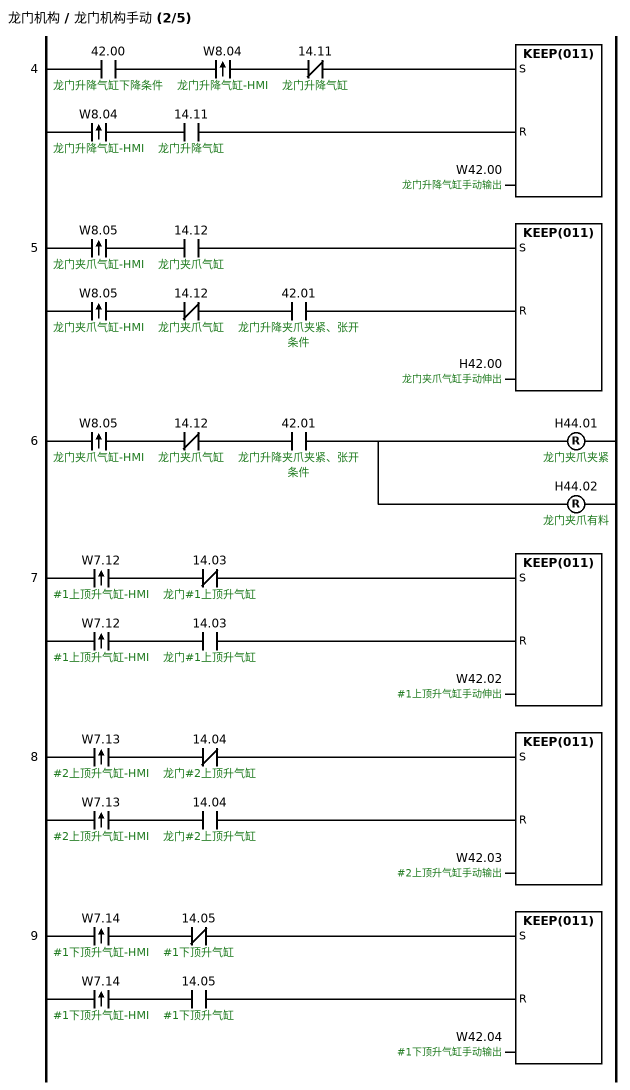
; [picture p377: 龙门机构 / 龙门机构手动, rungs 4-9]
; rung 4
LD 42.00  ; 龙门升降气缸下降条件
@AND W8.04  ; 龙门升降气缸-HMI
ANDNOT 14.11  ; 龙门升降气缸
@LD W8.04  ; 龙门升降气缸-HMI
AND 14.11  ; 龙门升降气缸
KEEP(011) W42.00  ; 龙门升降气缸手动输出
; rung 5
@LD W8.05  ; 龙门夹爪气缸-HMI
AND 14.12  ; 龙门夹爪气缸
@LD W8.05  ; 龙门夹爪气缸-HMI
ANDNOT 14.12  ; 龙门夹爪气缸
AND 42.01  ; 龙门升降夹爪夹紧、张开条件
KEEP(011) H42.00  ; 龙门夹爪气缸手动伸出
; rung 6
@LD W8.05  ; 龙门夹爪气缸-HMI
ANDNOT 14.12  ; 龙门夹爪气缸
AND 42.01  ; 龙门升降夹爪夹紧、张开条件
RSET H44.01  ; 龙门夹爪夹紧
RSET H44.02  ; 龙门夹爪有料
; rung 7
@LD W7.12  ; #1上顶升气缸-HMI
ANDNOT 14.03  ; 龙门#1上顶升气缸
@LD W7.12  ; #1上顶升气缸-HMI
AND 14.03  ; 龙门#1上顶升气缸
KEEP(011) W42.02  ; #1上顶升气缸手动伸出
; rung 8
@LD W7.13  ; #2上顶升气缸-HMI
ANDNOT 14.04  ; 龙门#2上顶升气缸
@LD W7.13  ; #2上顶升气缸-HMI
AND 14.04  ; 龙门#2上顶升气缸
KEEP(011) W42.03  ; #2上顶升气缸手动输出
; rung 9
@LD W7.14  ; #1下顶升气缸-HMI
ANDNOT 14.05  ; #1下顶升气缸
@LD W7.14  ; #1下顶升气缸-HMI
AND 14.05  ; #1下顶升气缸
KEEP(011) W42.04  ; #1下顶升气缸手动输出

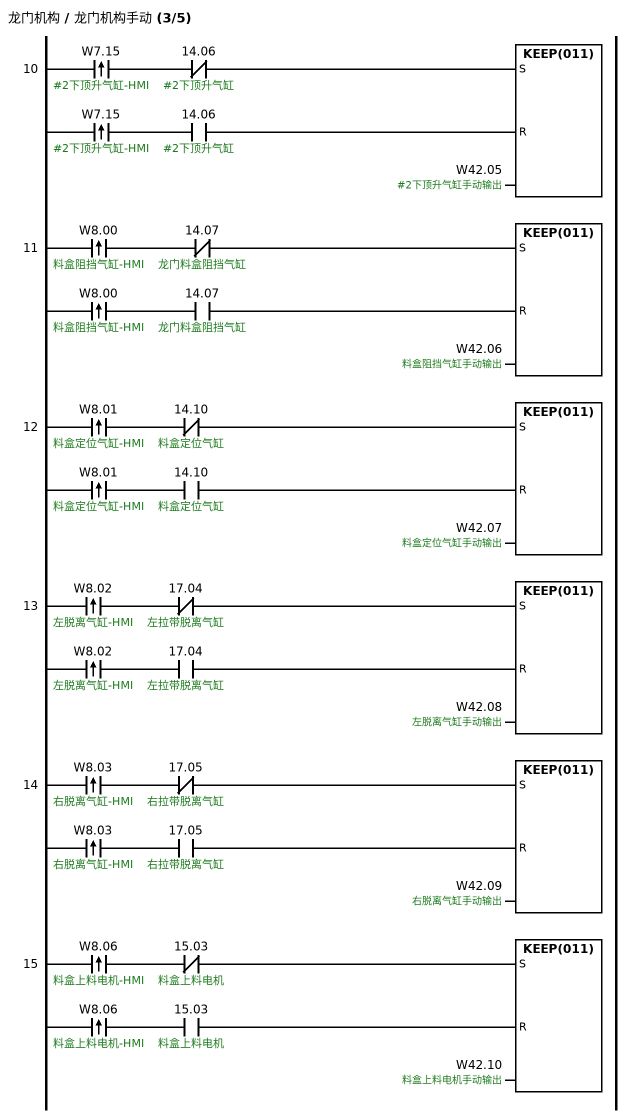
; rung 10
@LD W7.15  ; #2下顶升气缸-HMI
ANDNOT 14.06  ; #2下顶升气缸
@LD W7.15  ; #2下顶升气缸-HMI
AND 14.06  ; #2下顶升气缸
KEEP(011) W42.05  ; #2下顶升气缸手动输出
; rung 11
@LD W8.00  ; 料盒阻挡气缸-HMI
ANDNOT 14.07  ; 龙门料盒阻挡气缸
@LD W8.00  ; 料盒阻挡气缸-HMI
AND 14.07  ; 龙门料盒阻挡气缸
KEEP(011) W42.06  ; 料盒阻挡气缸手动输出
; rung 12
@LD W8.01  ; 料盒定位气缸-HMI
ANDNOT 14.10  ; 料盒定位气缸
@LD W8.01  ; 料盒定位气缸-HMI
AND 14.10  ; 料盒定位气缸
KEEP(011) W42.07  ; 料盒定位气缸手动输出
; rung 13
@LD W8.02  ; 左脱离气缸-HMI
ANDNOT 17.04  ; 左拉带脱离气缸
@LD W8.02  ; 左脱离气缸-HMI
AND 17.04  ; 左拉带脱离气缸
KEEP(011) W42.08  ; 左脱离气缸手动输出
; rung 14
@LD W8.03  ; 右脱离气缸-HMI
ANDNOT 17.05  ; 右拉带脱离气缸
@LD W8.03  ; 右脱离气缸-HMI
AND 17.05  ; 右拉带脱离气缸
KEEP(011) W42.09  ; 右脱离气缸手动输出
; rung 15
@LD W8.06  ; 料盒上料电机-HMI
ANDNOT 15.03  ; 料盒上料电机
@LD W8.06  ; 料盒上料电机-HMI
AND 15.03  ; 料盒上料电机
KEEP(011) W42.10  ; 料盒上料电机手动输出

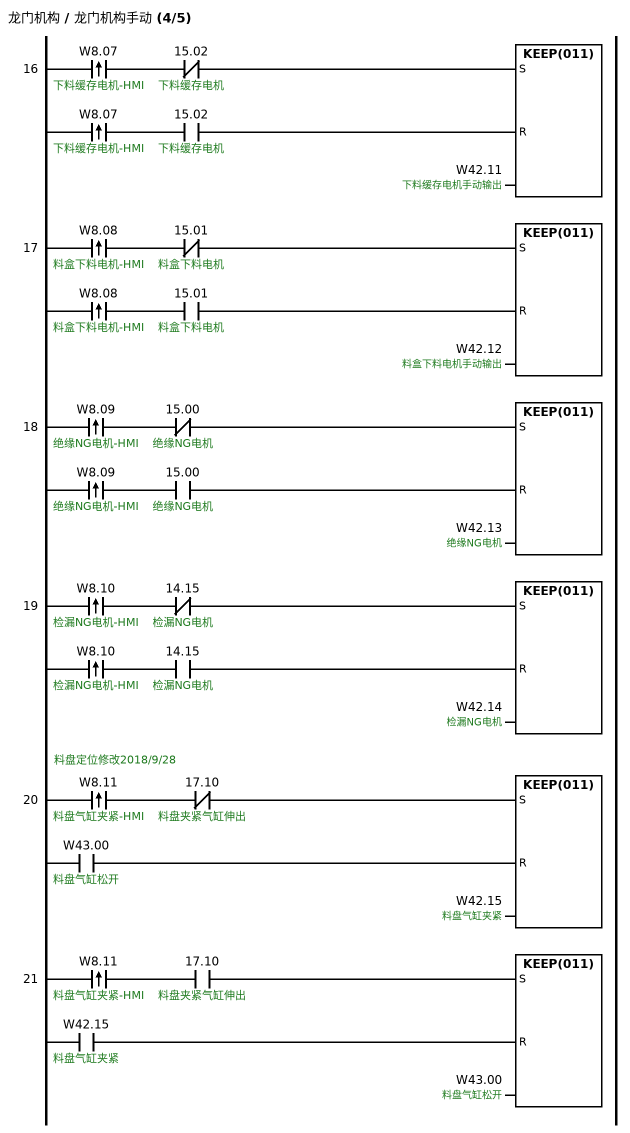
; rung 16
@LD W8.07  ; 下料缓存电机-HMI
ANDNOT 15.02  ; 下料缓存电机
@LD W8.07  ; 下料缓存电机-HMI
AND 15.02  ; 下料缓存电机
KEEP(011) W42.11  ; 下料缓存电机手动输出
; rung 17
@LD W8.08  ; 料盒下料电机-HMI
ANDNOT 15.01  ; 料盒下料电机
@LD W8.08  ; 料盒下料电机-HMI
AND 15.01  ; 料盒下料电机
KEEP(011) W42.12  ; 料盒下料电机手动输出
; rung 18
@LD W8.09  ; 绝缘NG电机-HMI
ANDNOT 15.00  ; 绝缘NG电机
@LD W8.09  ; 绝缘NG电机-HMI
AND 15.00  ; 绝缘NG电机
KEEP(011) W42.13  ; 绝缘NG电机
; rung 19
@LD W8.10  ; 检漏NG电机-HMI
ANDNOT 14.15  ; 检漏NG电机
@LD W8.10  ; 检漏NG电机-HMI
AND 14.15  ; 检漏NG电机
KEEP(011) W42.14  ; 检漏NG电机
; rung 20: 料盘定位修改2018/9/28
@LD W8.11  ; 料盘气缸夹紧-HMI
ANDNOT 17.10  ; 料盘夹紧气缸伸出
LD W43.00  ; 料盘气缸松开
KEEP(011) W42.15  ; 料盘气缸夹紧
; rung 21
@LD W8.11  ; 料盘气缸夹紧-HMI
AND 17.10  ; 料盘夹紧气缸伸出
LD W42.15  ; 料盘气缸夹紧
KEEP(011) W43.00  ; 料盘气缸松开

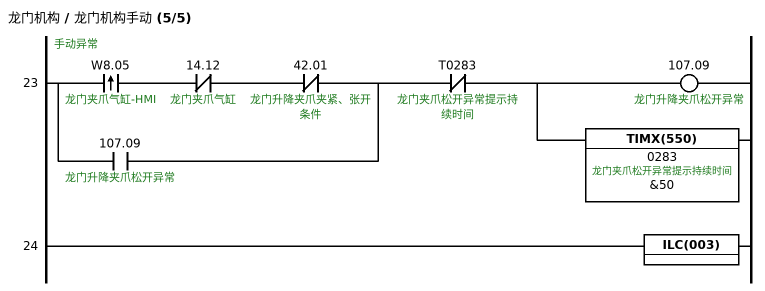
; rung 23: 手动异常
@LD W8.05  ; 龙门夹爪气缸-HMI
ANDNOT 14.12  ; 龙门夹爪气缸
ANDNOT 42.01  ; 龙门升降夹爪夹紧、张开条件
OR 107.09  ; 龙门升降夹爪松开异常
ANDNOT T0283  ; 龙门夹爪松开异常提示持续时间
OUT 107.09  ; 龙门升降夹爪松开异常
TIMX(550) 0283 &50  ; 龙门夹爪松开异常提示持续时间
; rung 24
ILC(003)

### Section 上料盒自动

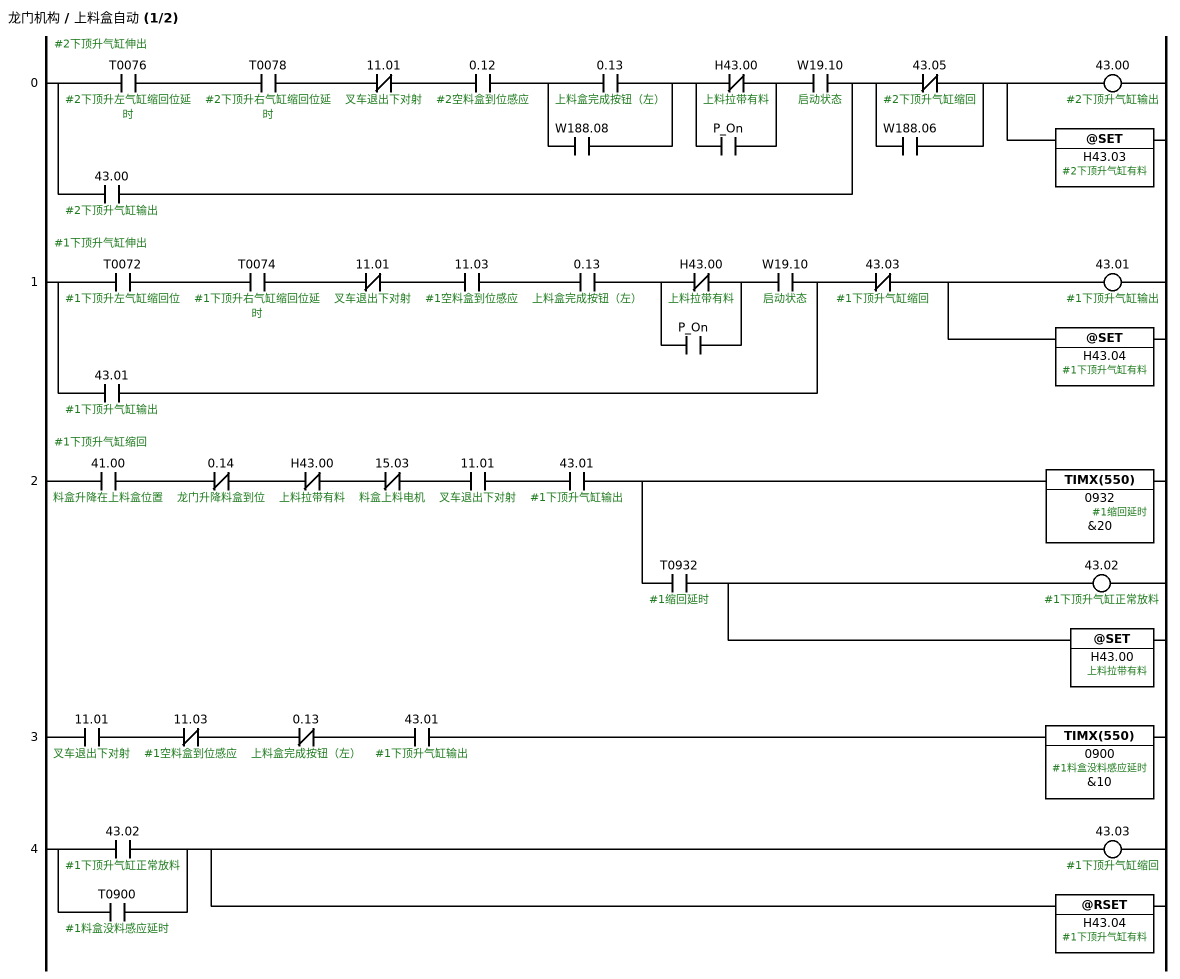
; rung 0: #2下顶升气缸伸出
LD T0076  ; #2下顶升左气缸缩回位延时
AND T0078  ; #2下顶升右气缸缩回位延时
ANDNOT 11.01  ; 叉车退出下对射
AND 0.12  ; #2空料盒到位感应
LD 0.13  ; 上料盒完成按钮（左）
OR W188.08
ANDLD
LDNOT H43.00  ; 上料拉带有料
OR P_On
ANDLD
AND W19.10  ; 启动状态
OR 43.00  ; #2下顶升气缸输出
LDNOT 43.05  ; #2下顶升气缸缩回
OR W188.06
ANDLD
OUT 43.00  ; #2下顶升气缸输出
@SET H43.03  ; #2下顶升气缸有料
; rung 1: #1下顶升气缸伸出
LD T0072  ; #1下顶升左气缸缩回位
AND T0074  ; #1下顶升右气缸缩回位延时
ANDNOT 11.01  ; 叉车退出下对射
AND 11.03  ; #1空料盒到位感应
AND 0.13  ; 上料盒完成按钮（左）
LDNOT H43.00  ; 上料拉带有料
OR P_On
ANDLD
AND W19.10  ; 启动状态
OR 43.01  ; #1下顶升气缸输出
ANDNOT 43.03  ; #1下顶升气缸缩回
OUT 43.01  ; #1下顶升气缸输出
@SET H43.04  ; #1下顶升气缸有料
; rung 2: #1下顶升气缸缩回
LD 41.00  ; 料盒升降在上料盒位置
ANDNOT 0.14  ; 龙门升降料盒到位
ANDNOT H43.00  ; 上料拉带有料
ANDNOT 15.03  ; 料盒上料电机
AND 11.01  ; 叉车退出下对射
AND 43.01  ; #1下顶升气缸输出
TIMX(550) 0932 &20  ; #1缩回延时
AND T0932  ; #1缩回延时
OUT 43.02  ; #1下顶升气缸正常放料
@SET H43.00  ; 上料拉带有料
; rung 3
LD 11.01  ; 叉车退出下对射
ANDNOT 11.03  ; #1空料盒到位感应
ANDNOT 0.13  ; 上料盒完成按钮（左）
AND 43.01  ; #1下顶升气缸输出
TIMX(550) 0900 &10  ; #1料盒没料感应延时
; rung 4
LD 43.02  ; #1下顶升气缸正常放料
OR T0900  ; #1料盒没料感应延时
OUT 43.03  ; #1下顶升气缸缩回
@RSET H43.04  ; #1下顶升气缸有料

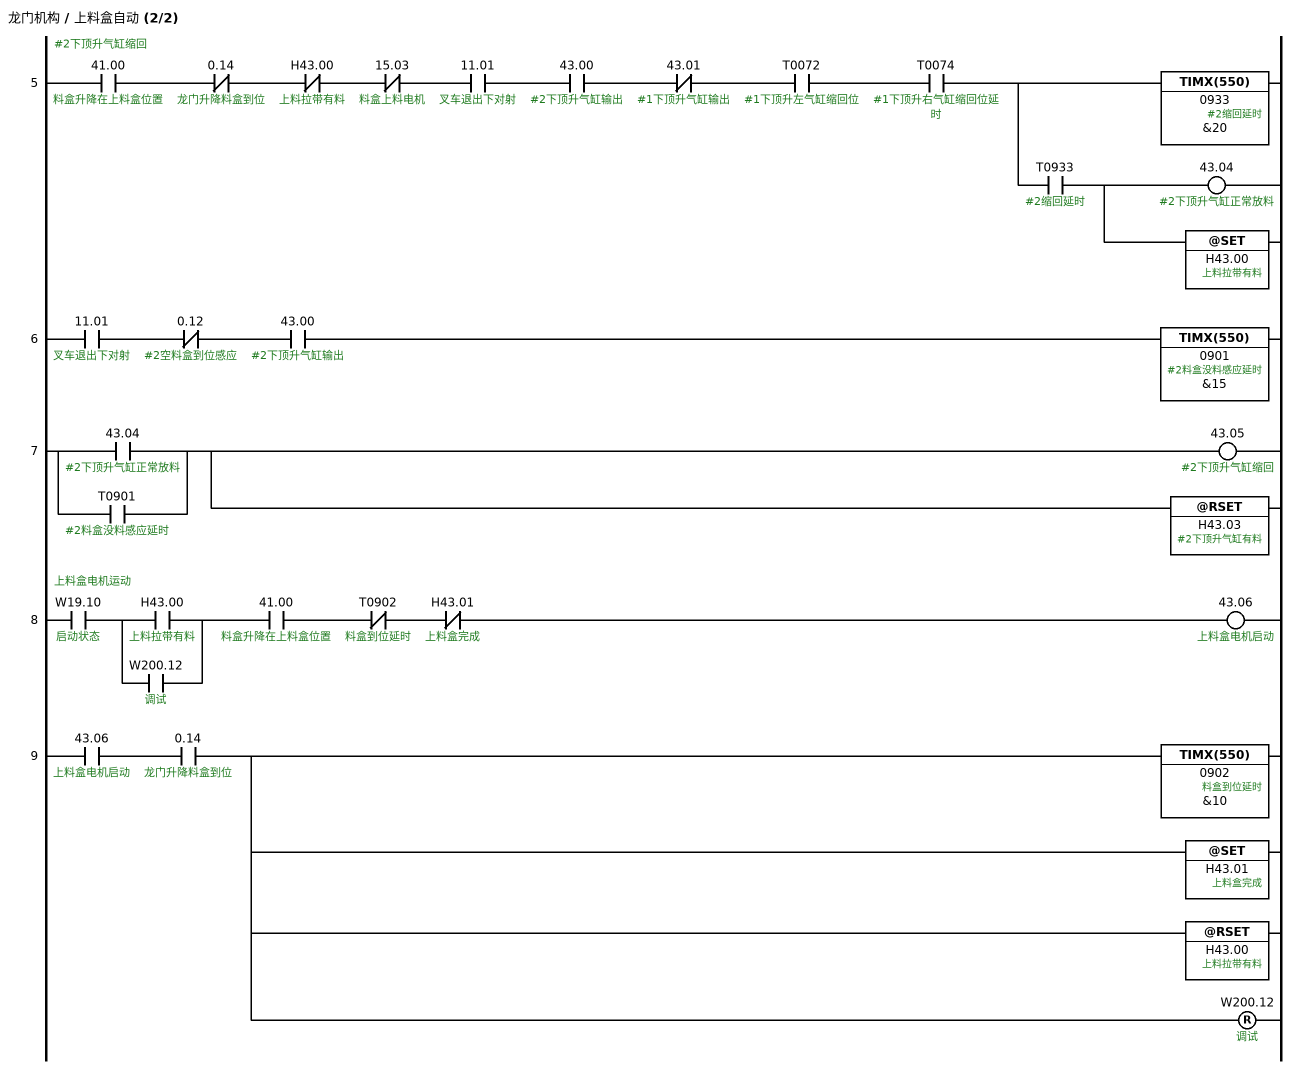
; rung 5: #2下顶升气缸缩回
LD 41.00  ; 料盒升降在上料盒位置
ANDNOT 0.14  ; 龙门升降料盒到位
ANDNOT H43.00  ; 上料拉带有料
ANDNOT 15.03  ; 料盒上料电机
AND 11.01  ; 叉车退出下对射
AND 43.00  ; #2下顶升气缸输出
ANDNOT 43.01  ; #1下顶升气缸输出
AND T0072  ; #1下顶升左气缸缩回位
AND T0074  ; #1下顶升右气缸缩回位延时
TIMX(550) 0933 &20  ; #2缩回延时
AND T0933  ; #2缩回延时
OUT 43.04  ; #2下顶升气缸正常放料
@SET H43.00  ; 上料拉带有料
; rung 6
LD 11.01  ; 叉车退出下对射
ANDNOT 0.12  ; #2空料盒到位感应
AND 43.00  ; #2下顶升气缸输出
TIMX(550) 0901 &15  ; #2料盒没料感应延时
; rung 7
LD 43.04  ; #2下顶升气缸正常放料
OR T0901  ; #2料盒没料感应延时
OUT 43.05  ; #2下顶升气缸缩回
@RSET H43.03  ; #2下顶升气缸有料
; rung 8: 上料盒电机运动
LD W19.10  ; 启动状态
LD H43.00  ; 上料拉带有料
OR W200.12  ; 调试
ANDLD
AND 41.00  ; 料盒升降在上料盒位置
ANDNOT T0902  ; 料盒到位延时
ANDNOT H43.01  ; 上料盒完成
OUT 43.06  ; 上料盒电机启动
; rung 9
LD 43.06  ; 上料盒电机启动
AND 0.14  ; 龙门升降料盒到位
TIMX(550) 0902 &10  ; 料盒到位延时
@SET H43.01  ; 上料盒完成
@RSET H43.00  ; 上料拉带有料
RSET W200.12  ; 调试

### Section 龙门机械手自动取放料

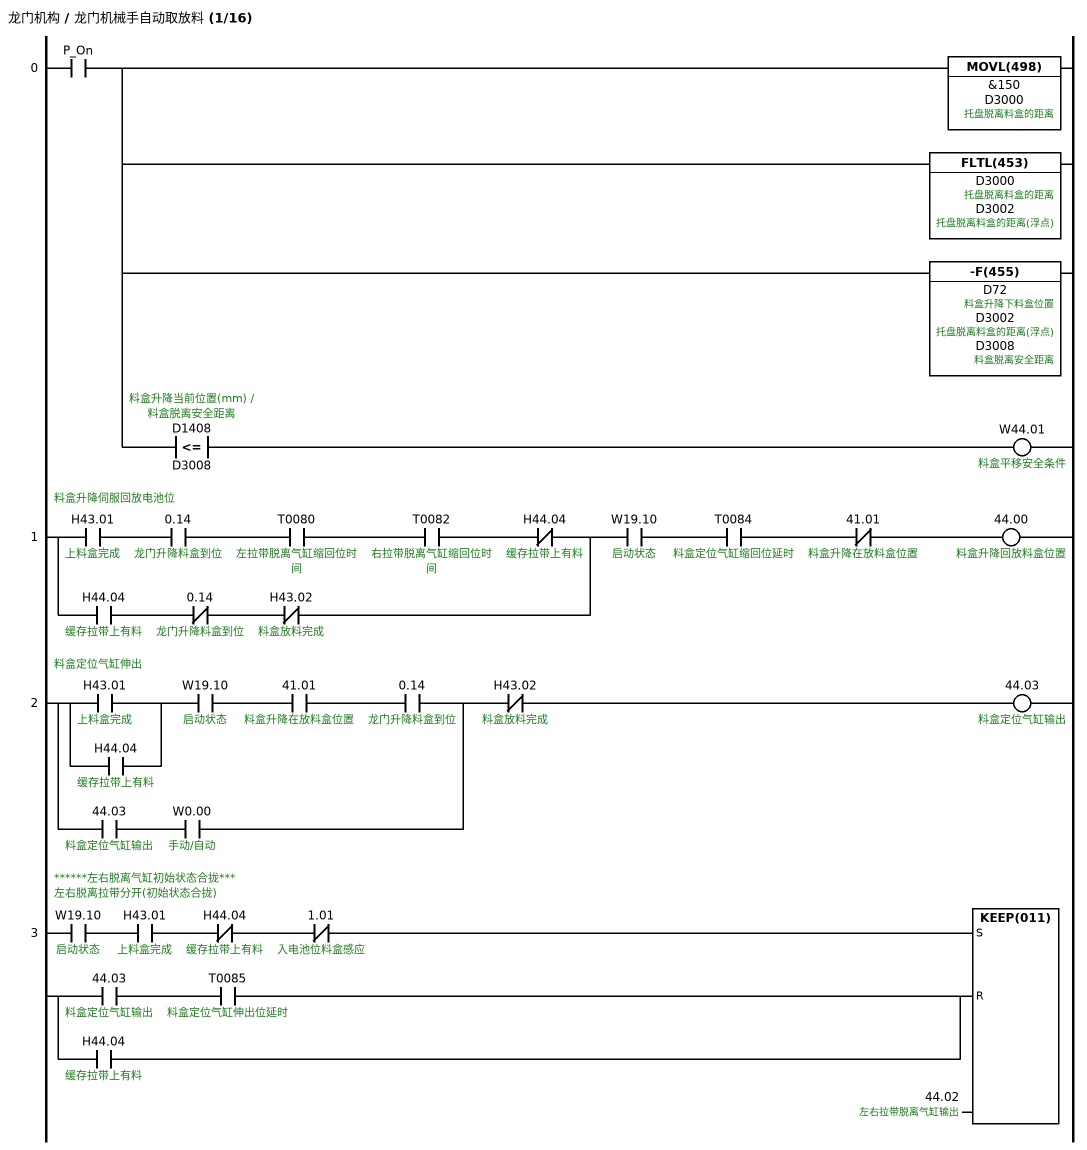
; rung 0
LD P_On
MOVL(498) &150 D3000  ; 托盘脱离料盒的距离
FLTL(453) D3000 D3002  ; 托盘脱离料盒的距离, 托盘脱离料盒的距离(浮点)
-F(455) D72 D3002 D3008  ; 料盒升降下料盒位置, 托盘脱离料盒的距离(浮点), 料盒脱离安全距离
AND<=F(332) D1408 D3008  ; 料盒升降当前位置(mm), 料盒脱离安全距离
OUT W44.01  ; 料盒平移安全条件
; rung 1: 料盒升降伺服回放电池位
LD H43.01  ; 上料盒完成
AND 0.14  ; 龙门升降料盒到位
AND T0080  ; 左拉带脱离气缸缩回位时间
AND T0082  ; 右拉带脱离气缸缩回位时间
ANDNOT H44.04  ; 缓存拉带上有料
LD H44.04  ; 缓存拉带上有料
ANDNOT 0.14  ; 龙门升降料盒到位
ANDNOT H43.02  ; 料盒放料完成
ORLD
AND W19.10  ; 启动状态
AND T0084  ; 料盒定位气缸缩回位延时
ANDNOT 41.01  ; 料盒升降在放料盒位置
OUT 44.00  ; 料盒升降回放料盒位置
; rung 2: 料盒定位气缸伸出
LD H43.01  ; 上料盒完成
OR H44.04  ; 缓存拉带上有料
AND W19.10  ; 启动状态
AND 41.01  ; 料盒升降在放料盒位置
AND 0.14  ; 龙门升降料盒到位
LD 44.03  ; 料盒定位气缸输出
AND W0.00  ; 手动/自动
ORLD
ANDNOT H43.02  ; 料盒放料完成
OUT 44.03  ; 料盒定位气缸输出
; rung 3: ******左右脱离气缸初始状态合拢*** / 左右脱离拉带分开(初始状态合拢)
LD W19.10  ; 启动状态
AND H43.01  ; 上料盒完成
ANDNOT H44.04  ; 缓存拉带上有料
ANDNOT 1.01  ; 入电池位料盒感应
LD 44.03  ; 料盒定位气缸输出
AND T0085  ; 料盒定位气缸伸出位延时
OR H44.04  ; 缓存拉带上有料
KEEP(011) 44.02  ; 左右拉带脱离气缸输出

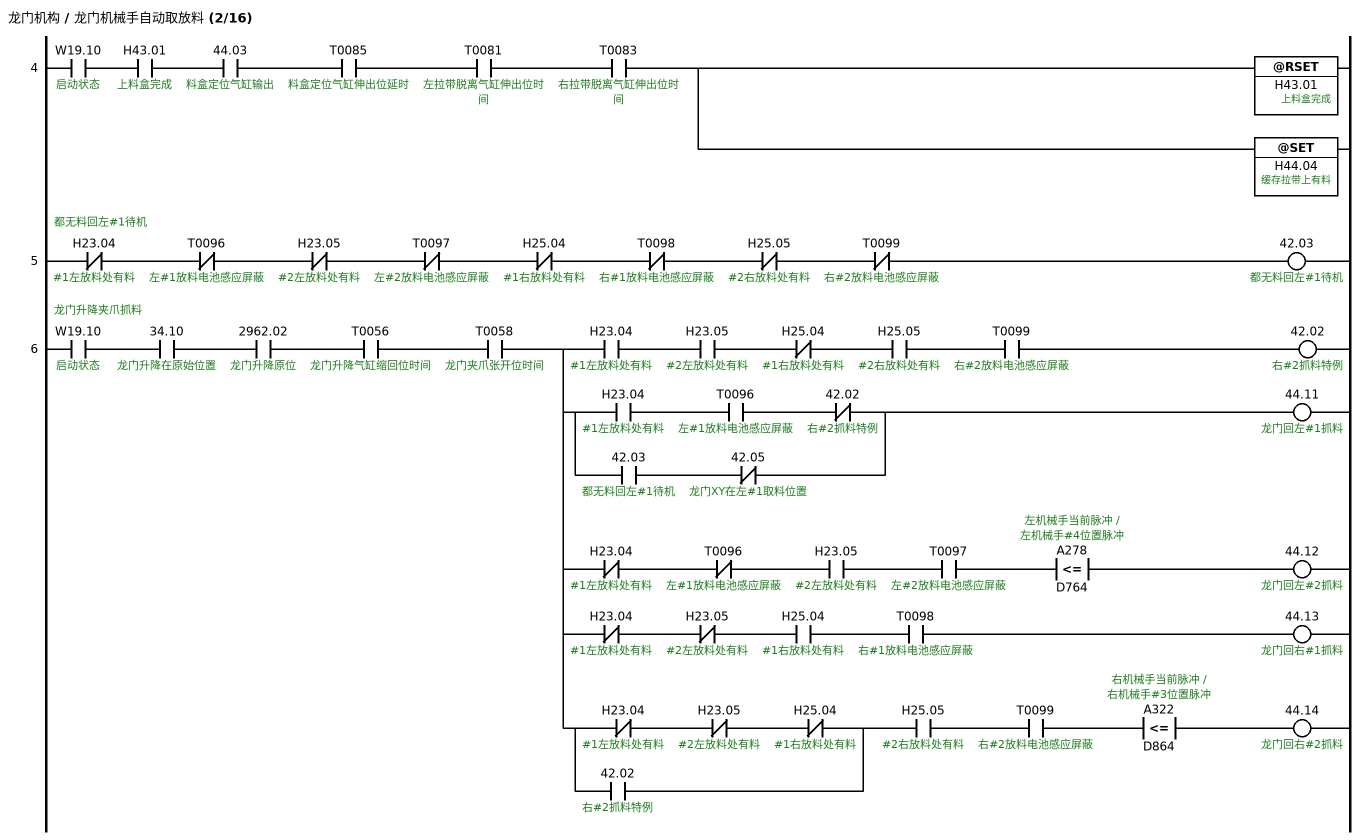
; rung 4
LD W19.10  ; 启动状态
AND H43.01  ; 上料盒完成
AND 44.03  ; 料盒定位气缸输出
AND T0085  ; 料盒定位气缸伸出位延时
AND T0081  ; 左拉带脱离气缸伸出位时间
AND T0083  ; 右拉带脱离气缸伸出位时间
@RSET H43.01  ; 上料盒完成
@SET H44.04  ; 缓存拉带上有料
; rung 5: 都无料回左#1待机
LDNOT H23.04  ; #1左放料处有料
ANDNOT T0096  ; 左#1放料电池感应屏蔽
ANDNOT H23.05  ; #2左放料处有料
ANDNOT T0097  ; 左#2放料电池感应屏蔽
ANDNOT H25.04  ; #1右放料处有料
ANDNOT T0098  ; 右#1放料电池感应屏蔽
ANDNOT H25.05  ; #2右放料处有料
ANDNOT T0099  ; 右#2放料电池感应屏蔽
OUT 42.03  ; 都无料回左#1待机
; rung 6: 龙门升降夹爪抓料
LD W19.10  ; 启动状态
AND 34.10  ; 龙门升降在原始位置
AND 2962.02  ; 龙门升降原位
AND T0056  ; 龙门升降气缸缩回位时间
AND T0058  ; 龙门夹爪张开位时间
OUT TR0
AND H23.04  ; #1左放料处有料
AND H23.05  ; #2左放料处有料
ANDNOT H25.04  ; #1右放料处有料
AND H25.05  ; #2右放料处有料
AND T0099  ; 右#2放料电池感应屏蔽
OUT 42.02  ; 右#2抓料特例
LD TR0
LD H23.04  ; #1左放料处有料
AND T0096  ; 左#1放料电池感应屏蔽
ANDNOT 42.02  ; 右#2抓料特例
LD 42.03  ; 都无料回左#1待机
ANDNOT 42.05  ; 龙门XY在左#1取料位置
ORLD
ANDLD
OUT 44.11  ; 龙门回左#1抓料
LD TR0
ANDNOT H23.04  ; #1左放料处有料
ANDNOT T0096  ; 左#1放料电池感应屏蔽
AND H23.05  ; #2左放料处有料
AND T0097  ; 左#2放料电池感应屏蔽
AND<=SL(318) A278 D764  ; 左机械手当前脉冲, 左机械手#4位置脉冲
OUT 44.12  ; 龙门回左#2抓料
LD TR0
ANDNOT H23.04  ; #1左放料处有料
ANDNOT H23.05  ; #2左放料处有料
AND H25.04  ; #1右放料处有料
AND T0098  ; 右#1放料电池感应屏蔽
OUT 44.13  ; 龙门回右#1抓料
LD TR0
LDNOT H23.04  ; #1左放料处有料
ANDNOT H23.05  ; #2左放料处有料
ANDNOT H25.04  ; #1右放料处有料
OR 42.02  ; 右#2抓料特例
ANDLD
AND H25.05  ; #2右放料处有料
AND T0099  ; 右#2放料电池感应屏蔽
AND<=SL(318) A322 D864  ; 右机械手当前脉冲, 右机械手#3位置脉冲
OUT 44.14  ; 龙门回右#2抓料

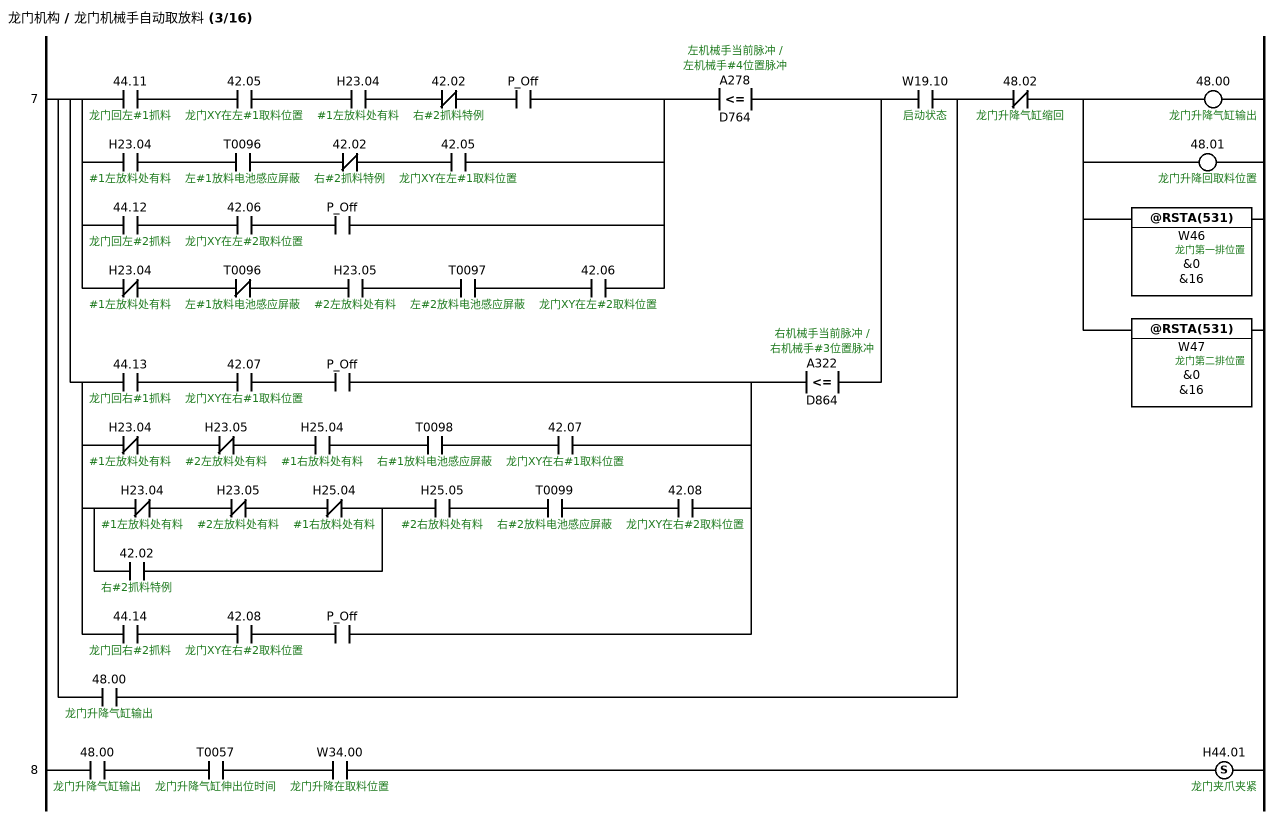
; rung 7
LD 44.11  ; 龙门回左#1抓料
AND 42.05  ; 龙门XY在左#1取料位置
AND H23.04  ; #1左放料处有料
ANDNOT 42.02  ; 右#2抓料特例
AND P_Off
LD H23.04  ; #1左放料处有料
AND T0096  ; 左#1放料电池感应屏蔽
ANDNOT 42.02  ; 右#2抓料特例
AND 42.05  ; 龙门XY在左#1取料位置
ORLD
LD 44.12  ; 龙门回左#2抓料
AND 42.06  ; 龙门XY在左#2取料位置
AND P_Off
ORLD
LDNOT H23.04  ; #1左放料处有料
ANDNOT T0096  ; 左#1放料电池感应屏蔽
AND H23.05  ; #2左放料处有料
AND T0097  ; 左#2放料电池感应屏蔽
AND 42.06  ; 龙门XY在左#2取料位置
ORLD
AND<=SL(318) A278 D764  ; 左机械手当前脉冲, 左机械手#4位置脉冲
LD 44.13  ; 龙门回右#1抓料
AND 42.07  ; 龙门XY在右#1取料位置
AND P_Off
LDNOT H23.04  ; #1左放料处有料
ANDNOT H23.05  ; #2左放料处有料
AND H25.04  ; #1右放料处有料
AND T0098  ; 右#1放料电池感应屏蔽
AND 42.07  ; 龙门XY在右#1取料位置
ORLD
LDNOT H23.04  ; #1左放料处有料
ANDNOT H23.05  ; #2左放料处有料
ANDNOT H25.04  ; #1右放料处有料
OR 42.02  ; 右#2抓料特例
AND H25.05  ; #2右放料处有料
AND T0099  ; 右#2放料电池感应屏蔽
AND 42.08  ; 龙门XY在右#2取料位置
ORLD
LD 44.14  ; 龙门回右#2抓料
AND 42.08  ; 龙门XY在右#2取料位置
AND P_Off
ORLD
AND<=SL(318) A322 D864  ; 右机械手当前脉冲, 右机械手#3位置脉冲
ORLD
AND W19.10  ; 启动状态
OR 48.00  ; 龙门升降气缸输出
ANDNOT 48.02  ; 龙门升降气缸缩回
OUT 48.00  ; 龙门升降气缸输出
OUT 48.01  ; 龙门升降回取料位置
@RSTA(531) W46 &0 &16  ; 龙门第一排位置
@RSTA(531) W47 &0 &16  ; 龙门第二排位置
; rung 8
LD 48.00  ; 龙门升降气缸输出
AND T0057  ; 龙门升降气缸伸出位时间
AND W34.00  ; 龙门升降在取料位置
SET H44.01  ; 龙门夹爪夹紧

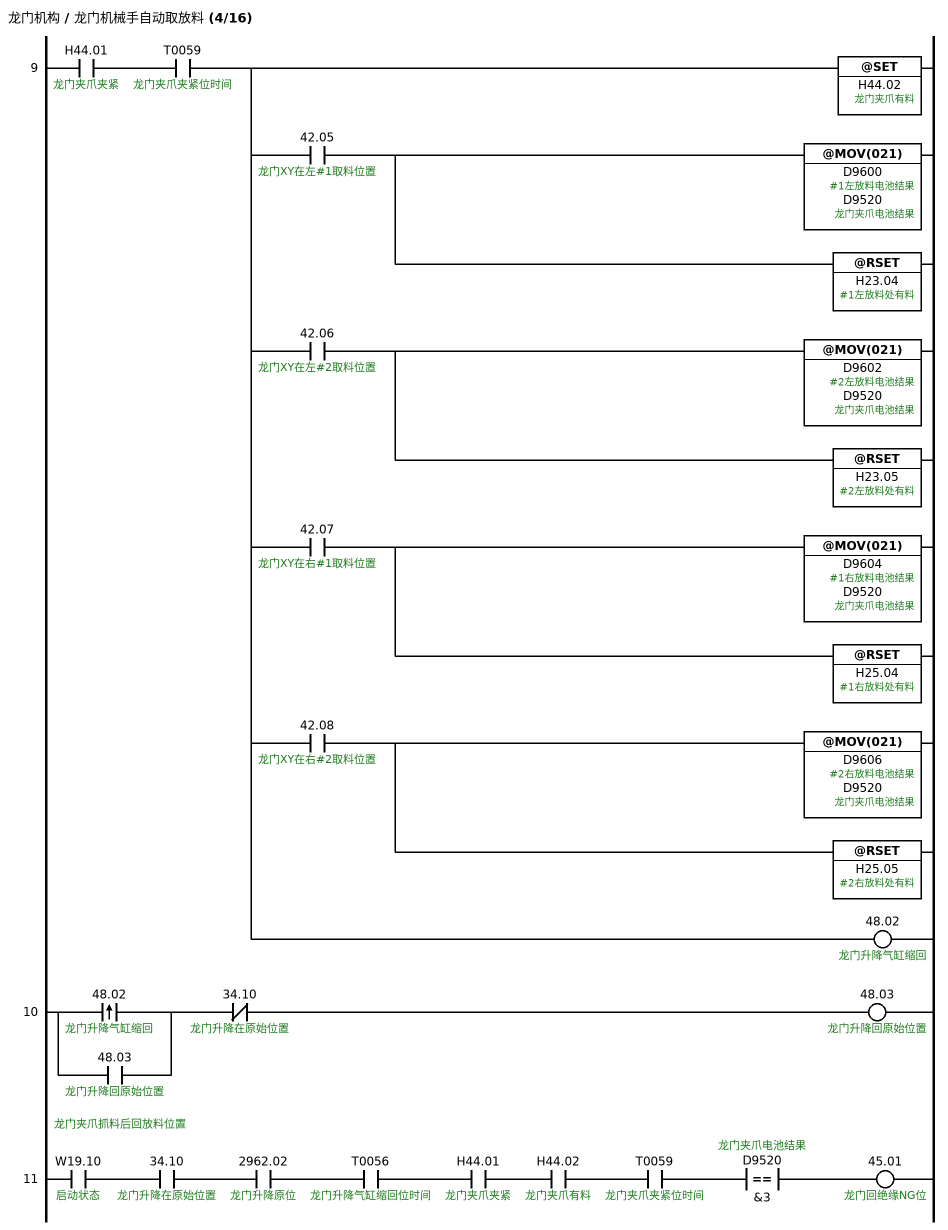
; rung 9
LD H44.01  ; 龙门夹爪夹紧
AND T0059  ; 龙门夹爪夹紧位时间
OUT TR0
@SET H44.02  ; 龙门夹爪有料
AND 42.05  ; 龙门XY在左#1取料位置
@MOV(021) D9600 D9520  ; #1左放料电池结果, 龙门夹爪电池结果
@RSET H23.04  ; #1左放料处有料
LD TR0
AND 42.06  ; 龙门XY在左#2取料位置
@MOV(021) D9602 D9520  ; #2左放料电池结果, 龙门夹爪电池结果
@RSET H23.05  ; #2左放料处有料
LD TR0
AND 42.07  ; 龙门XY在右#1取料位置
@MOV(021) D9604 D9520  ; #1右放料电池结果, 龙门夹爪电池结果
@RSET H25.04  ; #1右放料处有料
LD TR0
AND 42.08  ; 龙门XY在右#2取料位置
@MOV(021) D9606 D9520  ; #2右放料电池结果, 龙门夹爪电池结果
@RSET H25.05  ; #2右放料处有料
LD TR0
OUT 48.02  ; 龙门升降气缸缩回
; rung 10
@LD 48.02  ; 龙门升降气缸缩回
OR 48.03  ; 龙门升降回原始位置
ANDNOT 34.10  ; 龙门升降在原始位置
OUT 48.03  ; 龙门升降回原始位置
; rung 11: 龙门夹爪抓料后回放料位置
LD W19.10  ; 启动状态
AND 34.10  ; 龙门升降在原始位置
AND 2962.02  ; 龙门升降原位
AND T0056  ; 龙门升降气缸缩回位时间
AND H44.01  ; 龙门夹爪夹紧
AND H44.02  ; 龙门夹爪有料
AND T0059  ; 龙门夹爪夹紧位时间
AND=(300) D9520 &3  ; 龙门夹爪电池结果
OUT 45.01  ; 龙门回绝缘NG位

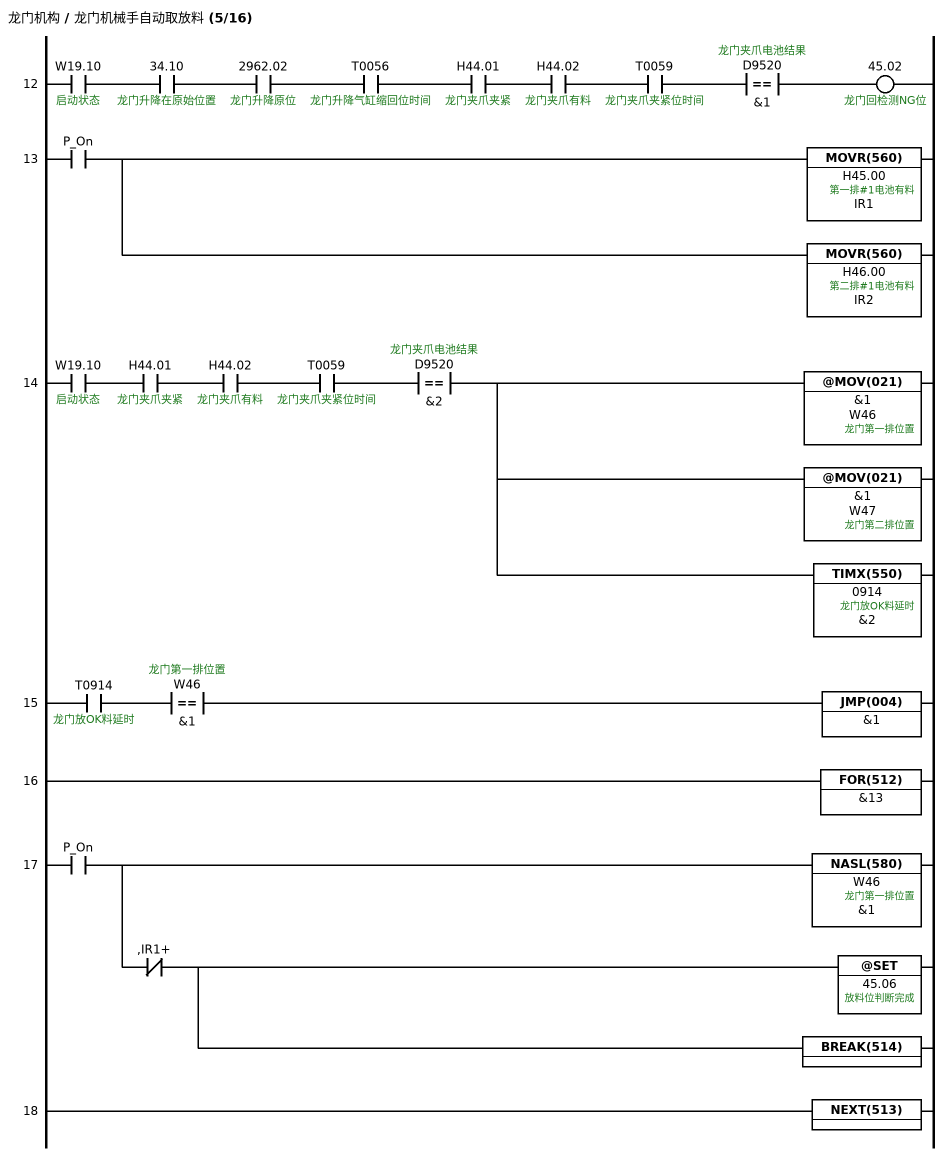
; rung 12
LD W19.10  ; 启动状态
AND 34.10  ; 龙门升降在原始位置
AND 2962.02  ; 龙门升降原位
AND T0056  ; 龙门升降气缸缩回位时间
AND H44.01  ; 龙门夹爪夹紧
AND H44.02  ; 龙门夹爪有料
AND T0059  ; 龙门夹爪夹紧位时间
AND=(300) D9520 &1  ; 龙门夹爪电池结果
OUT 45.02  ; 龙门回检测NG位
; rung 13
LD P_On
MOVR(560) H45.00 IR1  ; 第一排#1电池有料
MOVR(560) H46.00 IR2  ; 第二排#1电池有料
; rung 14
LD W19.10  ; 启动状态
AND H44.01  ; 龙门夹爪夹紧
AND H44.02  ; 龙门夹爪有料
AND T0059  ; 龙门夹爪夹紧位时间
AND=(300) D9520 &2  ; 龙门夹爪电池结果
@MOV(021) &1 W46  ; 龙门第一排位置
@MOV(021) &1 W47  ; 龙门第二排位置
TIMX(550) 0914 &2  ; 龙门放OK料延时
; rung 15
LD T0914  ; 龙门放OK料延时
AND=(300) W46 &1  ; 龙门第一排位置
JMP(004) &1
; rung 16
FOR(512) &13
; rung 17
LD P_On
NASL(580) W46 &1  ; 龙门第一排位置
ANDNOT ,IR1+
@SET 45.06  ; 放料位判断完成
BREAK(514)
; rung 18
NEXT(513)

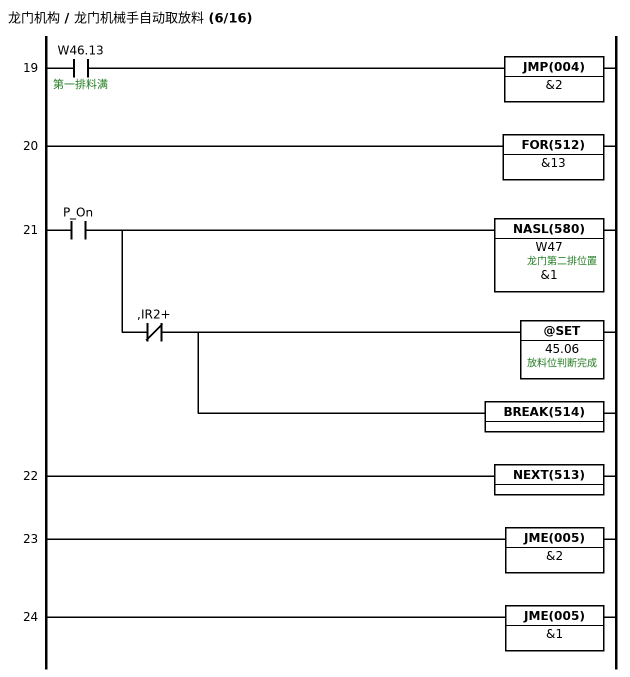
; rung 19
LD W46.13  ; 第一排料满
JMP(004) &2
; rung 20
FOR(512) &13
; rung 21
LD P_On
NASL(580) W47 &1  ; 龙门第二排位置
ANDNOT ,IR2+
@SET 45.06  ; 放料位判断完成
BREAK(514)
; rung 22
NEXT(513)
; rung 23
JME(005) &2
; rung 24
JME(005) &1

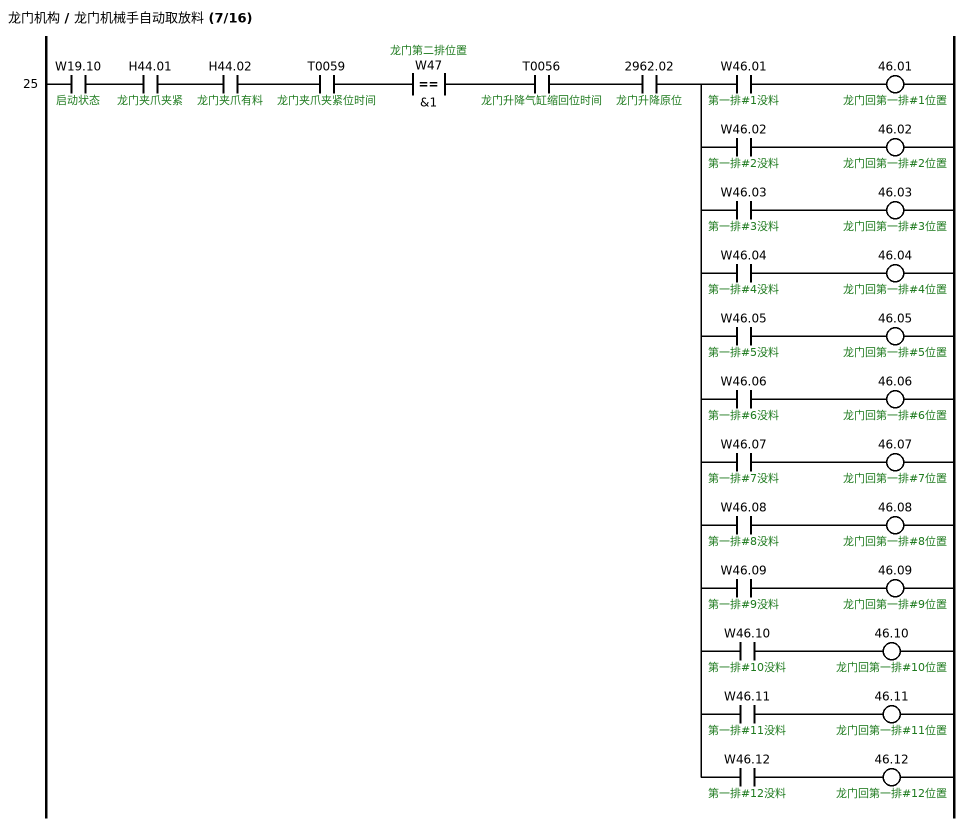
; rung 25
LD W19.10  ; 启动状态
AND H44.01  ; 龙门夹爪夹紧
AND H44.02  ; 龙门夹爪有料
AND T0059  ; 龙门夹爪夹紧位时间
AND=(300) W47 &1  ; 龙门第二排位置
AND T0056  ; 龙门升降气缸缩回位时间
AND 2962.02  ; 龙门升降原位
OUT TR0
AND W46.01  ; 第一排#1没料
OUT 46.01  ; 龙门回第一排#1位置
LD TR0
AND W46.02  ; 第一排#2没料
OUT 46.02  ; 龙门回第一排#2位置
LD TR0
AND W46.03  ; 第一排#3没料
OUT 46.03  ; 龙门回第一排#3位置
LD TR0
AND W46.04  ; 第一排#4没料
OUT 46.04  ; 龙门回第一排#4位置
LD TR0
AND W46.05  ; 第一排#5没料
OUT 46.05  ; 龙门回第一排#5位置
LD TR0
AND W46.06  ; 第一排#6没料
OUT 46.06  ; 龙门回第一排#6位置
LD TR0
AND W46.07  ; 第一排#7没料
OUT 46.07  ; 龙门回第一排#7位置
LD TR0
AND W46.08  ; 第一排#8没料
OUT 46.08  ; 龙门回第一排#8位置
LD TR0
AND W46.09  ; 第一排#9没料
OUT 46.09  ; 龙门回第一排#9位置
LD TR0
AND W46.10  ; 第一排#10没料
OUT 46.10  ; 龙门回第一排#10位置
LD TR0
AND W46.11  ; 第一排#11没料
OUT 46.11  ; 龙门回第一排#11位置
LD TR0
AND W46.12  ; 第一排#12没料
OUT 46.12  ; 龙门回第一排#12位置

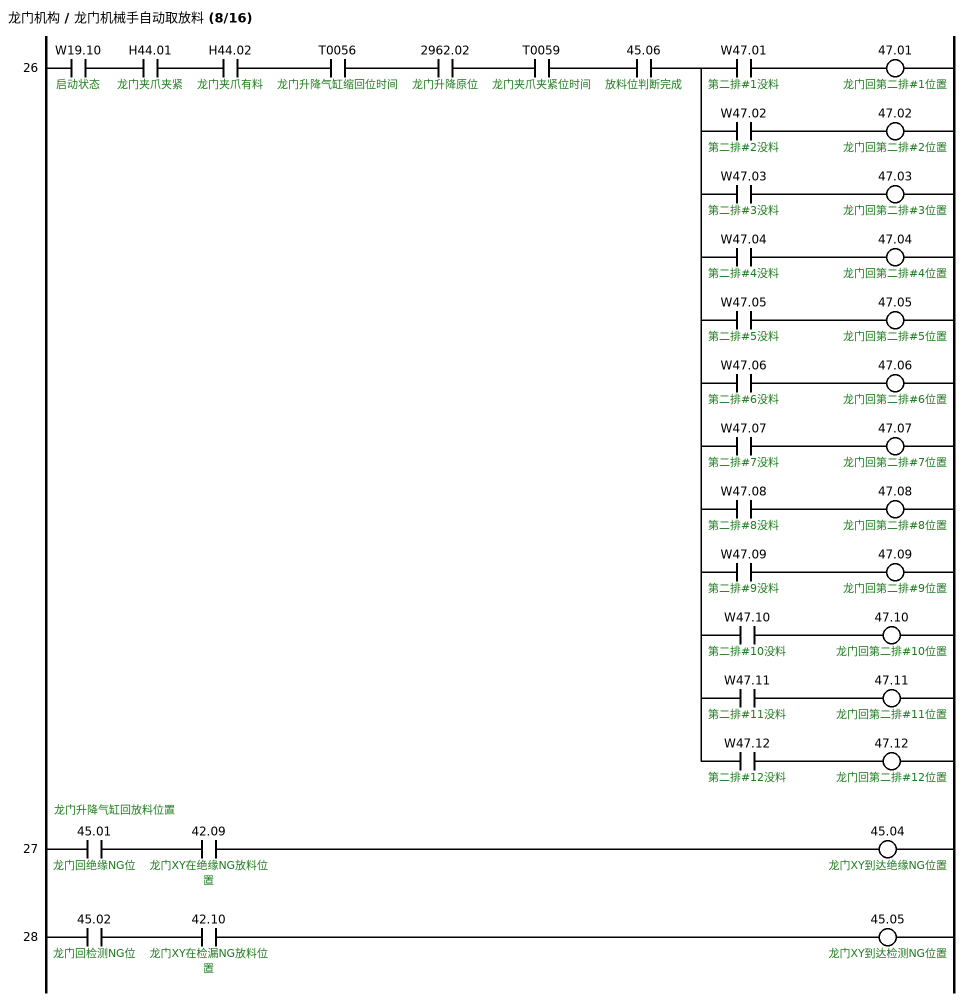
; rung 26
LD W19.10  ; 启动状态
AND H44.01  ; 龙门夹爪夹紧
AND H44.02  ; 龙门夹爪有料
AND T0056  ; 龙门升降气缸缩回位时间
AND 2962.02  ; 龙门升降原位
AND T0059  ; 龙门夹爪夹紧位时间
AND 45.06  ; 放料位判断完成
OUT TR0
AND W47.01  ; 第二排#1没料
OUT 47.01  ; 龙门回第二排#1位置
LD TR0
AND W47.02  ; 第二排#2没料
OUT 47.02  ; 龙门回第二排#2位置
LD TR0
AND W47.03  ; 第二排#3没料
OUT 47.03  ; 龙门回第二排#3位置
LD TR0
AND W47.04  ; 第二排#4没料
OUT 47.04  ; 龙门回第二排#4位置
LD TR0
AND W47.05  ; 第二排#5没料
OUT 47.05  ; 龙门回第二排#5位置
LD TR0
AND W47.06  ; 第二排#6没料
OUT 47.06  ; 龙门回第二排#6位置
LD TR0
AND W47.07  ; 第二排#7没料
OUT 47.07  ; 龙门回第二排#7位置
LD TR0
AND W47.08  ; 第二排#8没料
OUT 47.08  ; 龙门回第二排#8位置
LD TR0
AND W47.09  ; 第二排#9没料
OUT 47.09  ; 龙门回第二排#9位置
LD TR0
AND W47.10  ; 第二排#10没料
OUT 47.10  ; 龙门回第二排#10位置
LD TR0
AND W47.11  ; 第二排#11没料
OUT 47.11  ; 龙门回第二排#11位置
LD TR0
AND W47.12  ; 第二排#12没料
OUT 47.12  ; 龙门回第二排#12位置
; rung 27: 龙门升降气缸回放料位置
LD 45.01  ; 龙门回绝缘NG位
AND 42.09  ; 龙门XY在绝缘NG放料位置
OUT 45.04  ; 龙门XY到达绝缘NG位置
; rung 28
LD 45.02  ; 龙门回检测NG位
AND 42.10  ; 龙门XY在检漏NG放料位置
OUT 45.05  ; 龙门XY到达检测NG位置

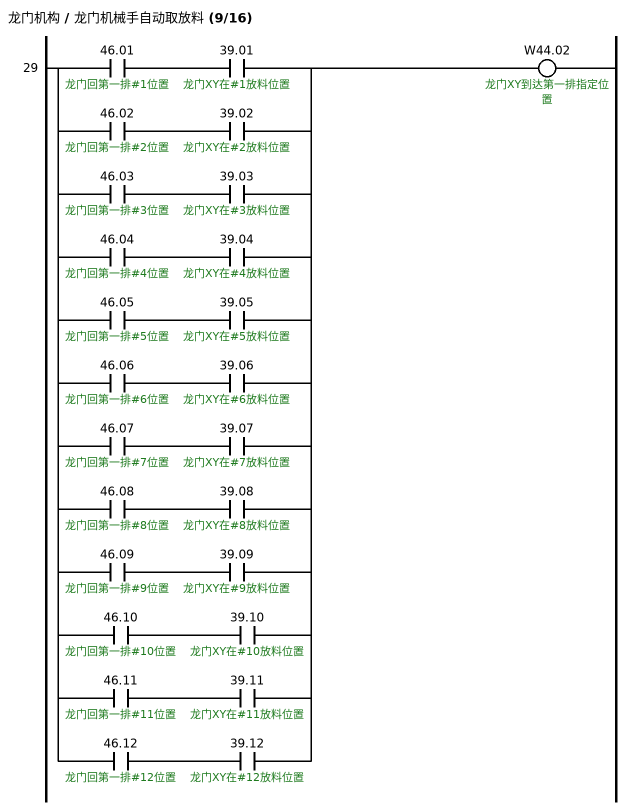
; rung 29
LD 46.01  ; 龙门回第一排#1位置
AND 39.01  ; 龙门XY在#1放料位置
LD 46.02  ; 龙门回第一排#2位置
AND 39.02  ; 龙门XY在#2放料位置
ORLD
LD 46.03  ; 龙门回第一排#3位置
AND 39.03  ; 龙门XY在#3放料位置
ORLD
LD 46.04  ; 龙门回第一排#4位置
AND 39.04  ; 龙门XY在#4放料位置
ORLD
LD 46.05  ; 龙门回第一排#5位置
AND 39.05  ; 龙门XY在#5放料位置
ORLD
LD 46.06  ; 龙门回第一排#6位置
AND 39.06  ; 龙门XY在#6放料位置
ORLD
LD 46.07  ; 龙门回第一排#7位置
AND 39.07  ; 龙门XY在#7放料位置
ORLD
LD 46.08  ; 龙门回第一排#8位置
AND 39.08  ; 龙门XY在#8放料位置
ORLD
LD 46.09  ; 龙门回第一排#9位置
AND 39.09  ; 龙门XY在#9放料位置
ORLD
LD 46.10  ; 龙门回第一排#10位置
AND 39.10  ; 龙门XY在#10放料位置
ORLD
LD 46.11  ; 龙门回第一排#11位置
AND 39.11  ; 龙门XY在#11放料位置
ORLD
LD 46.12  ; 龙门回第一排#12位置
AND 39.12  ; 龙门XY在#12放料位置
ORLD
OUT W44.02  ; 龙门XY到达第一排指定位置

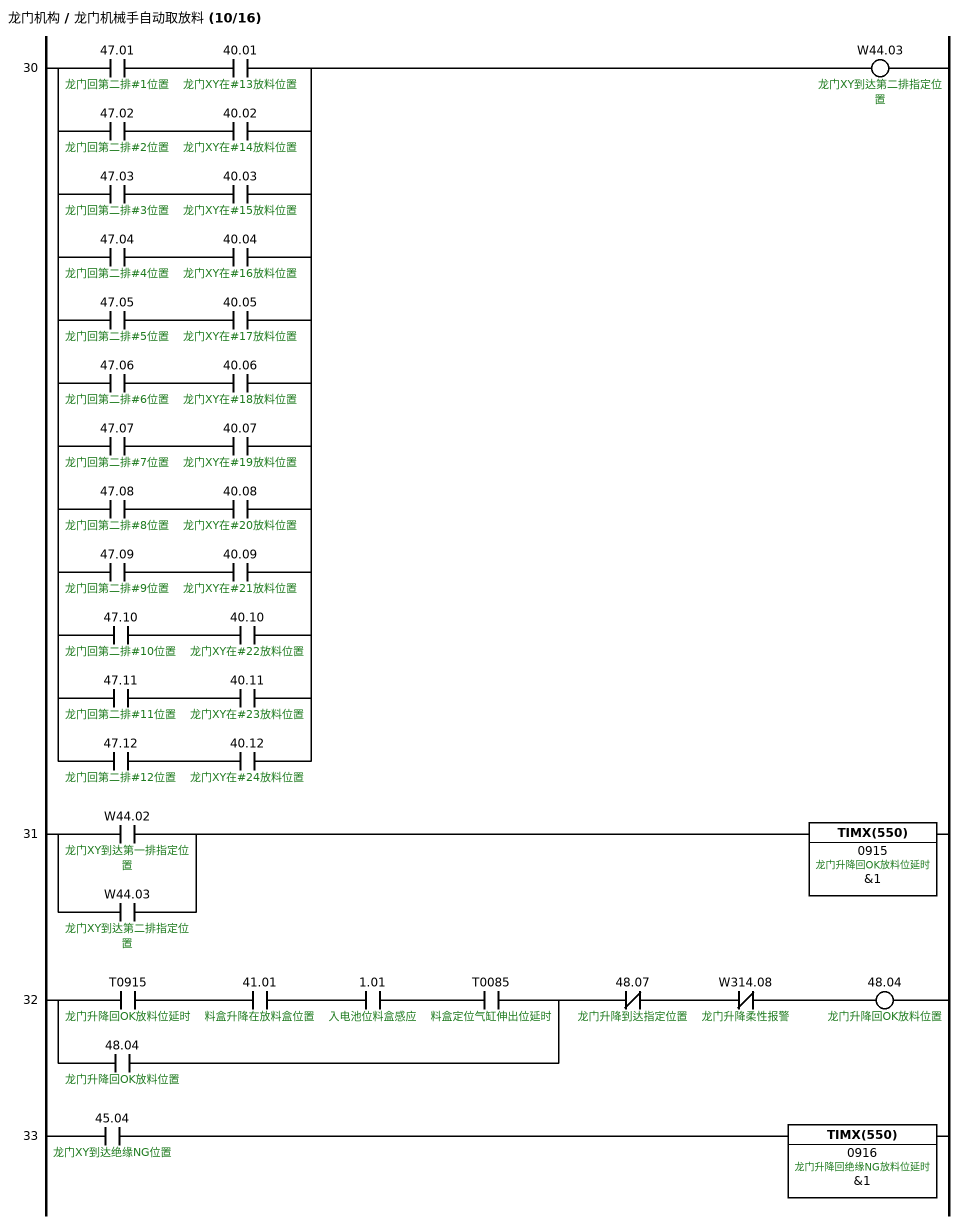
; rung 30
LD 47.01  ; 龙门回第二排#1位置
AND 40.01  ; 龙门XY在#13放料位置
LD 47.02  ; 龙门回第二排#2位置
AND 40.02  ; 龙门XY在#14放料位置
ORLD
LD 47.03  ; 龙门回第二排#3位置
AND 40.03  ; 龙门XY在#15放料位置
ORLD
LD 47.04  ; 龙门回第二排#4位置
AND 40.04  ; 龙门XY在#16放料位置
ORLD
LD 47.05  ; 龙门回第二排#5位置
AND 40.05  ; 龙门XY在#17放料位置
ORLD
LD 47.06  ; 龙门回第二排#6位置
AND 40.06  ; 龙门XY在#18放料位置
ORLD
LD 47.07  ; 龙门回第二排#7位置
AND 40.07  ; 龙门XY在#19放料位置
ORLD
LD 47.08  ; 龙门回第二排#8位置
AND 40.08  ; 龙门XY在#20放料位置
ORLD
LD 47.09  ; 龙门回第二排#9位置
AND 40.09  ; 龙门XY在#21放料位置
ORLD
LD 47.10  ; 龙门回第二排#10位置
AND 40.10  ; 龙门XY在#22放料位置
ORLD
LD 47.11  ; 龙门回第二排#11位置
AND 40.11  ; 龙门XY在#23放料位置
ORLD
LD 47.12  ; 龙门回第二排#12位置
AND 40.12  ; 龙门XY在#24放料位置
ORLD
OUT W44.03  ; 龙门XY到达第二排指定位置
; rung 31
LD W44.02  ; 龙门XY到达第一排指定位置
OR W44.03  ; 龙门XY到达第二排指定位置
TIMX(550) 0915 &1  ; 龙门升降回OK放料位延时
; rung 32
LD T0915  ; 龙门升降回OK放料位延时
AND 41.01  ; 料盒升降在放料盒位置
AND 1.01  ; 入电池位料盒感应
AND T0085  ; 料盒定位气缸伸出位延时
OR 48.04  ; 龙门升降回OK放料位置
ANDNOT 48.07  ; 龙门升降到达指定位置
ANDNOT W314.08  ; 龙门升降柔性报警
OUT 48.04  ; 龙门升降回OK放料位置
; rung 33
LD 45.04  ; 龙门XY到达绝缘NG位置
TIMX(550) 0916 &1  ; 龙门升降回绝缘NG放料位延时

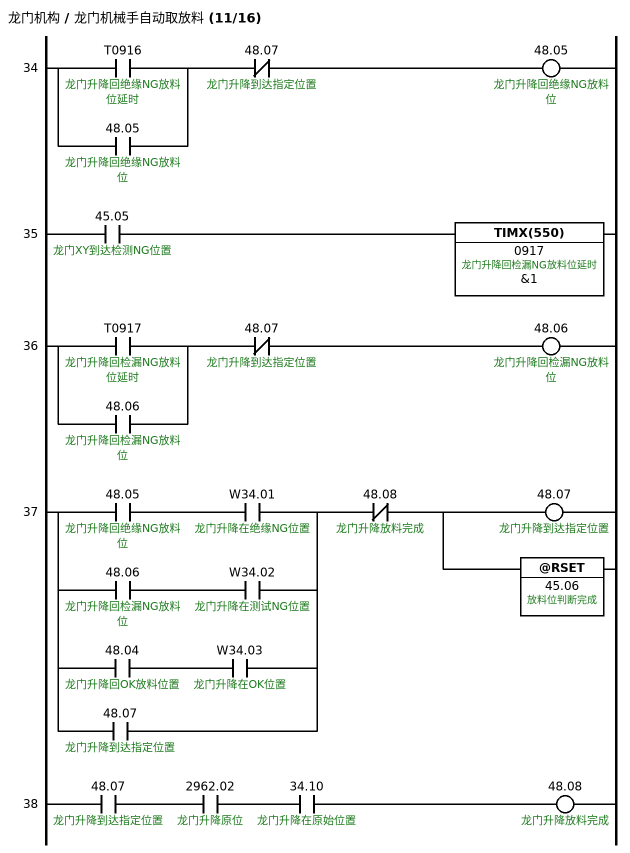
; rung 34
LD T0916  ; 龙门升降回绝缘NG放料位延时
OR 48.05  ; 龙门升降回绝缘NG放料位
ANDNOT 48.07  ; 龙门升降到达指定位置
OUT 48.05  ; 龙门升降回绝缘NG放料位
; rung 35
LD 45.05  ; 龙门XY到达检测NG位置
TIMX(550) 0917 &1  ; 龙门升降回检漏NG放料位延时
; rung 36
LD T0917  ; 龙门升降回检漏NG放料位延时
OR 48.06  ; 龙门升降回检漏NG放料位
ANDNOT 48.07  ; 龙门升降到达指定位置
OUT 48.06  ; 龙门升降回检漏NG放料位
; rung 37
LD 48.05  ; 龙门升降回绝缘NG放料位
AND W34.01  ; 龙门升降在绝缘NG位置
LD 48.06  ; 龙门升降回检漏NG放料位
AND W34.02  ; 龙门升降在测试NG位置
ORLD
LD 48.04  ; 龙门升降回OK放料位置
AND W34.03  ; 龙门升降在OK位置
ORLD
OR 48.07  ; 龙门升降到达指定位置
ANDNOT 48.08  ; 龙门升降放料完成
OUT 48.07  ; 龙门升降到达指定位置
@RSET 45.06  ; 放料位判断完成
; rung 38
LD 48.07  ; 龙门升降到达指定位置
AND 2962.02  ; 龙门升降原位
AND 34.10  ; 龙门升降在原始位置
OUT 48.08  ; 龙门升降放料完成

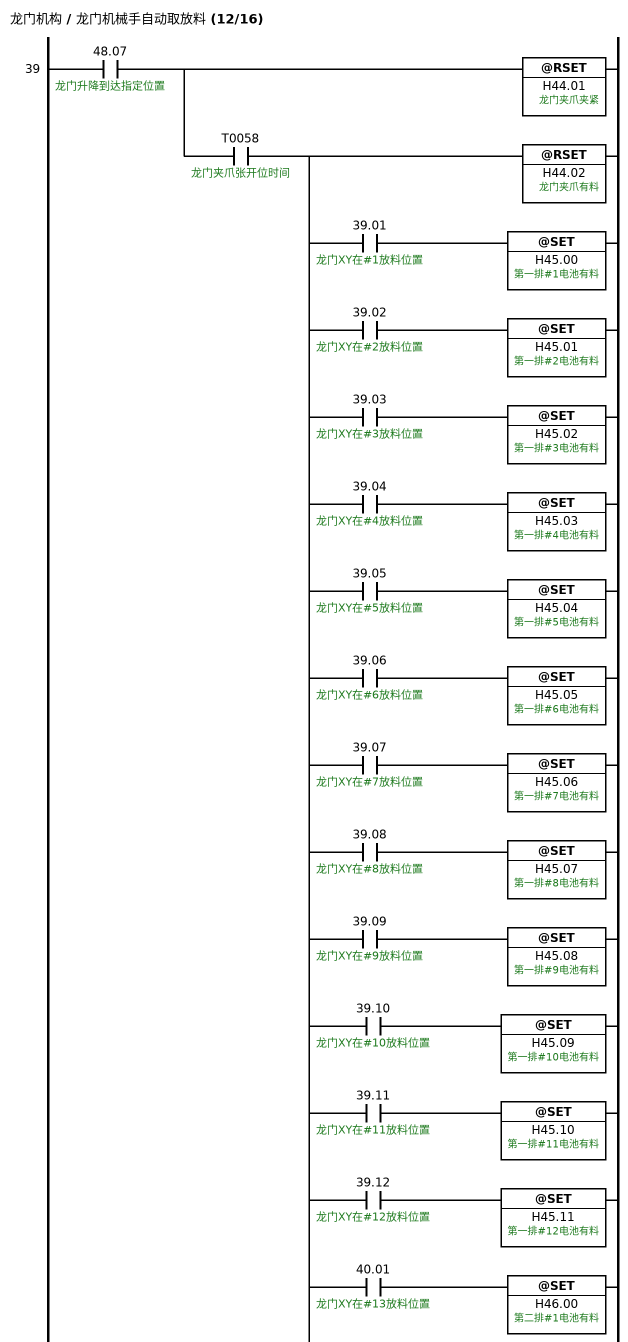

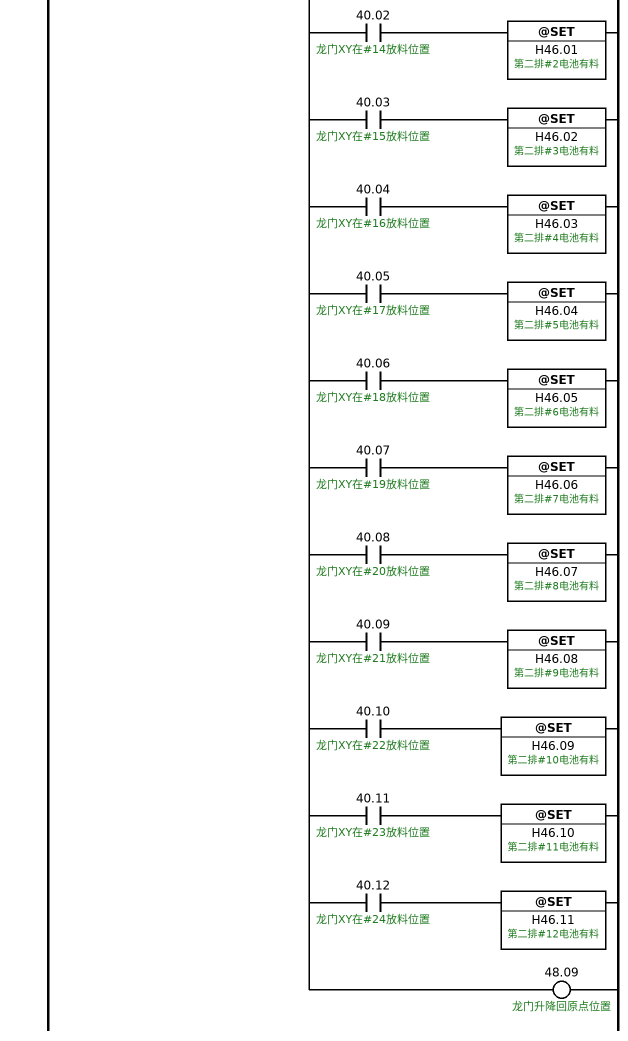
; rung 39
LD 48.07  ; 龙门升降到达指定位置
@RSET H44.01  ; 龙门夹爪夹紧
AND T0058  ; 龙门夹爪张开位时间
OUT TR0
@RSET H44.02  ; 龙门夹爪有料
AND 39.01  ; 龙门XY在#1放料位置
@SET H45.00  ; 第一排#1电池有料
LD TR0
AND 39.02  ; 龙门XY在#2放料位置
@SET H45.01  ; 第一排#2电池有料
LD TR0
AND 39.03  ; 龙门XY在#3放料位置
@SET H45.02  ; 第一排#3电池有料
LD TR0
AND 39.04  ; 龙门XY在#4放料位置
@SET H45.03  ; 第一排#4电池有料
LD TR0
AND 39.05  ; 龙门XY在#5放料位置
@SET H45.04  ; 第一排#5电池有料
LD TR0
AND 39.06  ; 龙门XY在#6放料位置
@SET H45.05  ; 第一排#6电池有料
LD TR0
AND 39.07  ; 龙门XY在#7放料位置
@SET H45.06  ; 第一排#7电池有料
LD TR0
AND 39.08  ; 龙门XY在#8放料位置
@SET H45.07  ; 第一排#8电池有料
LD TR0
AND 39.09  ; 龙门XY在#9放料位置
@SET H45.08  ; 第一排#9电池有料
LD TR0
AND 39.10  ; 龙门XY在#10放料位置
@SET H45.09  ; 第一排#10电池有料
LD TR0
AND 39.11  ; 龙门XY在#11放料位置
@SET H45.10  ; 第一排#11电池有料
LD TR0
AND 39.12  ; 龙门XY在#12放料位置
@SET H45.11  ; 第一排#12电池有料
LD TR0
AND 40.01  ; 龙门XY在#13放料位置
@SET H46.00  ; 第二排#1电池有料
LD TR0
AND 40.02  ; 龙门XY在#14放料位置
@SET H46.01  ; 第二排#2电池有料
LD TR0
AND 40.03  ; 龙门XY在#15放料位置
@SET H46.02  ; 第二排#3电池有料
LD TR0
AND 40.04  ; 龙门XY在#16放料位置
@SET H46.03  ; 第二排#4电池有料
LD TR0
AND 40.05  ; 龙门XY在#17放料位置
@SET H46.04  ; 第二排#5电池有料
LD TR0
AND 40.06  ; 龙门XY在#18放料位置
@SET H46.05  ; 第二排#6电池有料
LD TR0
AND 40.07  ; 龙门XY在#19放料位置
@SET H46.06  ; 第二排#7电池有料
LD TR0
AND 40.08  ; 龙门XY在#20放料位置
@SET H46.07  ; 第二排#8电池有料
LD TR0
AND 40.09  ; 龙门XY在#21放料位置
@SET H46.08  ; 第二排#9电池有料
LD TR0
AND 40.10  ; 龙门XY在#22放料位置
@SET H46.09  ; 第二排#10电池有料
LD TR0
AND 40.11  ; 龙门XY在#23放料位置
@SET H46.10  ; 第二排#11电池有料
LD TR0
AND 40.12  ; 龙门XY在#24放料位置
@SET H46.11  ; 第二排#12电池有料
LD TR0
OUT 48.09  ; 龙门升降回原点位置

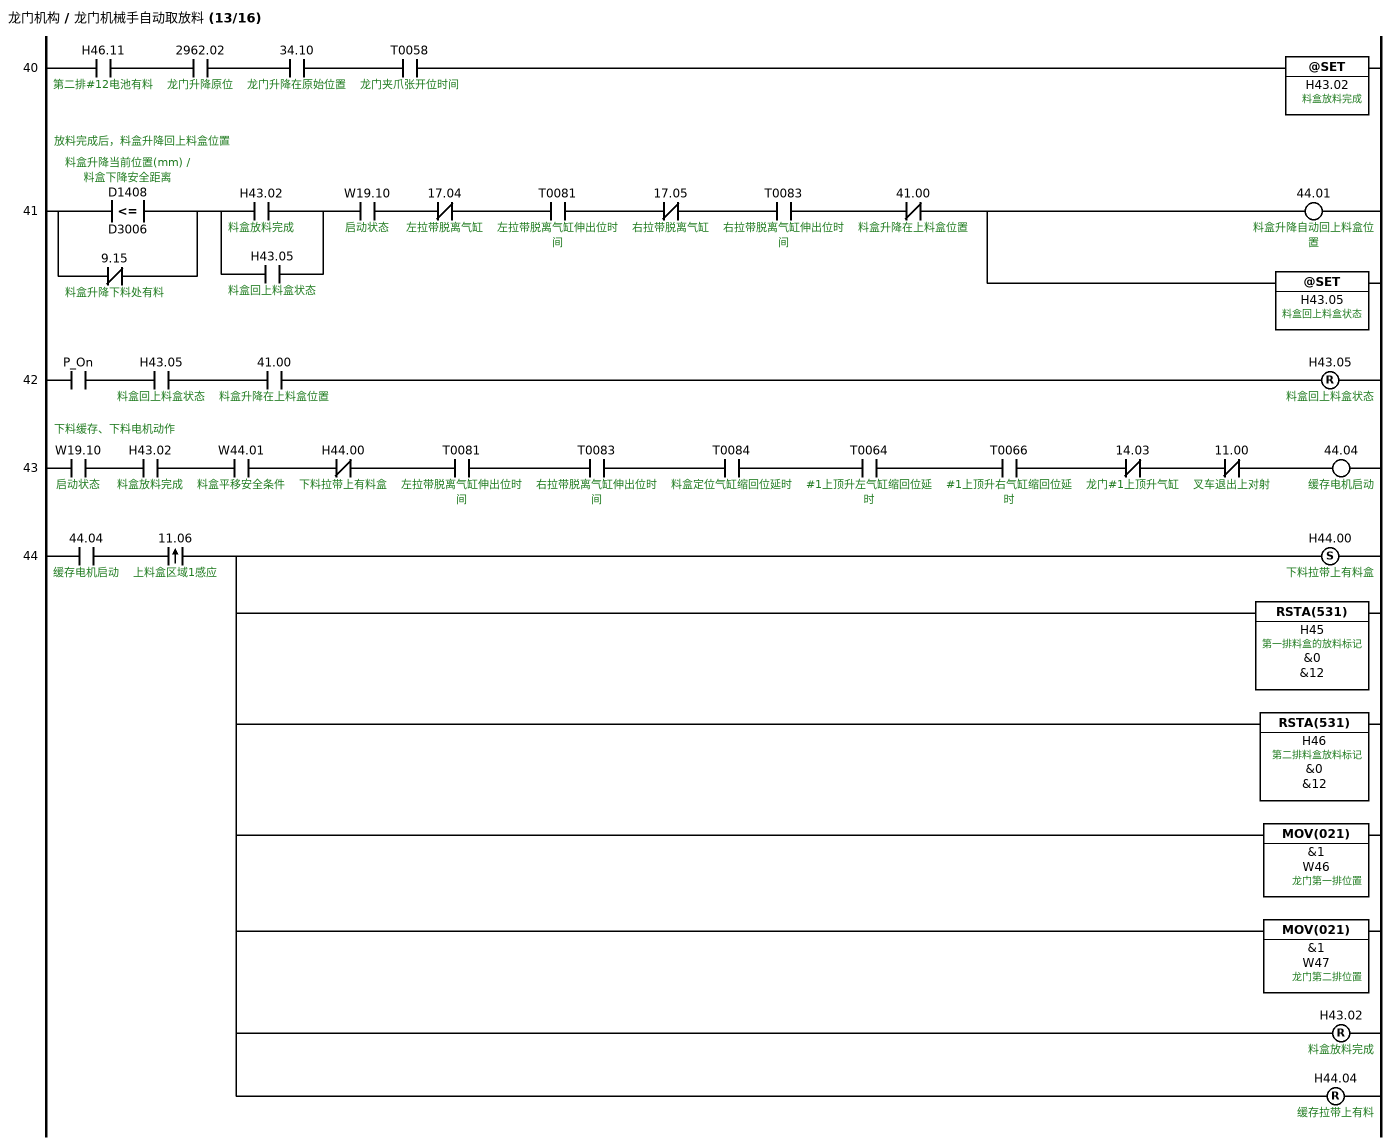
; rung 40
LD H46.11  ; 第二排#12电池有料
AND 2962.02  ; 龙门升降原位
AND 34.10  ; 龙门升降在原始位置
AND T0058  ; 龙门夹爪张开位时间
@SET H43.02  ; 料盒放料完成
; rung 41: 放料完成后，料盒升降回上料盒位置
LD<=F(332) D1408 D3006  ; 料盒升降当前位置(mm), 料盒下降安全距离
ORNOT 9.15  ; 料盒升降下料处有料
LD H43.02  ; 料盒放料完成
OR H43.05  ; 料盒回上料盒状态
ANDLD
AND W19.10  ; 启动状态
ANDNOT 17.04  ; 左拉带脱离气缸
AND T0081  ; 左拉带脱离气缸伸出位时间
ANDNOT 17.05  ; 右拉带脱离气缸
AND T0083  ; 右拉带脱离气缸伸出位时间
ANDNOT 41.00  ; 料盒升降在上料盒位置
OUT 44.01  ; 料盒升降自动回上料盒位置
@SET H43.05  ; 料盒回上料盒状态
; rung 42
LD P_On
AND H43.05  ; 料盒回上料盒状态
AND 41.00  ; 料盒升降在上料盒位置
RSET H43.05  ; 料盒回上料盒状态
; rung 43: 下料缓存、下料电机动作
LD W19.10  ; 启动状态
AND H43.02  ; 料盒放料完成
AND W44.01  ; 料盒平移安全条件
ANDNOT H44.00  ; 下料拉带上有料盒
AND T0081  ; 左拉带脱离气缸伸出位时间
AND T0083  ; 右拉带脱离气缸伸出位时间
AND T0084  ; 料盒定位气缸缩回位延时
AND T0064  ; #1上顶升左气缸缩回位延时
AND T0066  ; #1上顶升右气缸缩回位延时
ANDNOT 14.03  ; 龙门#1上顶升气缸
ANDNOT 11.00  ; 叉车退出上对射
OUT 44.04  ; 缓存电机启动
; rung 44
LD 44.04  ; 缓存电机启动
@AND 11.06  ; 上料盒区域1感应
SET H44.00  ; 下料拉带上有料盒
RSTA(531) H45 &0 &12  ; 第一排料盒的放料标记
RSTA(531) H46 &0 &12  ; 第二排料盒放料标记
MOV(021) &1 W46  ; 龙门第一排位置
MOV(021) &1 W47  ; 龙门第二排位置
RSET H43.02  ; 料盒放料完成
RSET H44.04  ; 缓存拉带上有料

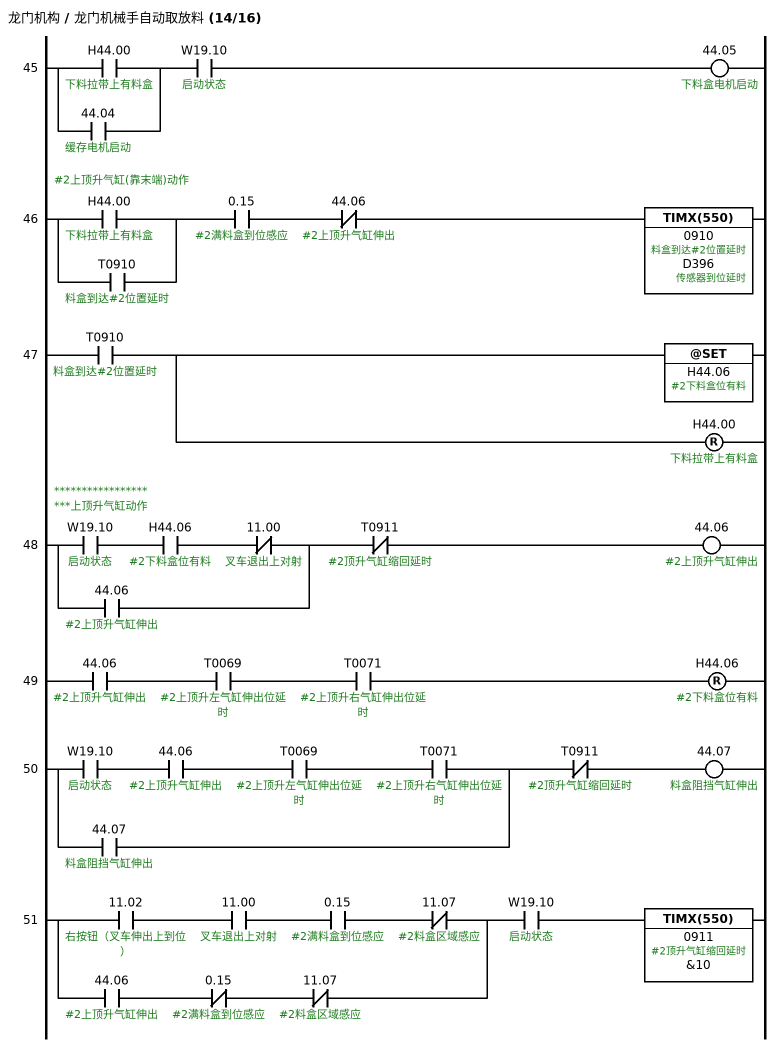
; rung 45
LD H44.00  ; 下料拉带上有料盒
OR 44.04  ; 缓存电机启动
AND W19.10  ; 启动状态
OUT 44.05  ; 下料盒电机启动
; rung 46: #2上顶升气缸(靠末端)动作
LD H44.00  ; 下料拉带上有料盒
OR T0910  ; 料盒到达#2位置延时
AND 0.15  ; #2满料盒到位感应
ANDNOT 44.06  ; #2上顶升气缸伸出
TIMX(550) 0910 D396  ; 传感器到位延时, 料盒到达#2位置延时
; rung 47
LD T0910  ; 料盒到达#2位置延时
@SET H44.06  ; #2下料盒位有料
RSET H44.00  ; 下料拉带上有料盒
; rung 48: ***************** / ***上顶升气缸动作
LD W19.10  ; 启动状态
AND H44.06  ; #2下料盒位有料
ANDNOT 11.00  ; 叉车退出上对射
OR 44.06  ; #2上顶升气缸伸出
ANDNOT T0911  ; #2顶升气缸缩回延时
OUT 44.06  ; #2上顶升气缸伸出
; rung 49
LD 44.06  ; #2上顶升气缸伸出
AND T0069  ; #2上顶升左气缸伸出位延时
AND T0071  ; #2上顶升右气缸伸出位延时
RSET H44.06  ; #2下料盒位有料
; rung 50
LD W19.10  ; 启动状态
AND 44.06  ; #2上顶升气缸伸出
AND T0069  ; #2上顶升左气缸伸出位延时
AND T0071  ; #2上顶升右气缸伸出位延时
OR 44.07  ; 料盒阻挡气缸伸出
ANDNOT T0911  ; #2顶升气缸缩回延时
OUT 44.07  ; 料盒阻挡气缸伸出
; rung 51
LD 11.02  ; 右按钮（叉车伸出上到位）
AND 11.00  ; 叉车退出上对射
AND 0.15  ; #2满料盒到位感应
ANDNOT 11.07  ; #2料盒区域感应
LD 44.06  ; #2上顶升气缸伸出
ANDNOT 0.15  ; #2满料盒到位感应
ANDNOT 11.07  ; #2料盒区域感应
ORLD
AND W19.10  ; 启动状态
TIMX(550) 0911 &10  ; #2顶升气缸缩回延时

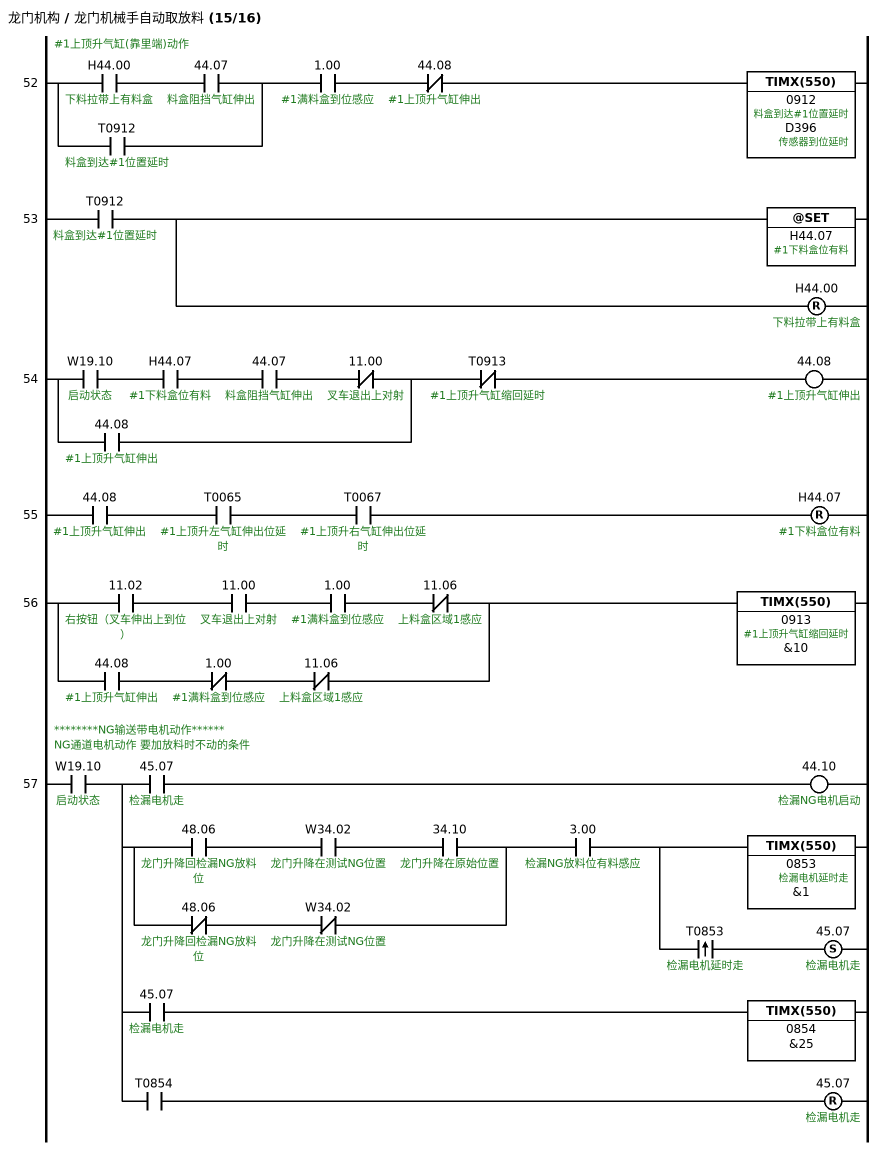
; rung 52: #1上顶升气缸(靠里端)动作
LD H44.00  ; 下料拉带上有料盒
AND 44.07  ; 料盒阻挡气缸伸出
OR T0912  ; 料盒到达#1位置延时
AND 1.00  ; #1满料盒到位感应
ANDNOT 44.08  ; #1上顶升气缸伸出
TIMX(550) 0912 D396  ; 传感器到位延时, 料盒到达#1位置延时
; rung 53
LD T0912  ; 料盒到达#1位置延时
@SET H44.07  ; #1下料盒位有料
RSET H44.00  ; 下料拉带上有料盒
; rung 54
LD W19.10  ; 启动状态
AND H44.07  ; #1下料盒位有料
AND 44.07  ; 料盒阻挡气缸伸出
ANDNOT 11.00  ; 叉车退出上对射
OR 44.08  ; #1上顶升气缸伸出
ANDNOT T0913  ; #1上顶升气缸缩回延时
OUT 44.08  ; #1上顶升气缸伸出
; rung 55
LD 44.08  ; #1上顶升气缸伸出
AND T0065  ; #1上顶升左气缸伸出位延时
AND T0067  ; #1上顶升右气缸伸出位延时
RSET H44.07  ; #1下料盒位有料
; rung 56
LD 11.02  ; 右按钮（叉车伸出上到位）
AND 11.00  ; 叉车退出上对射
AND 1.00  ; #1满料盒到位感应
ANDNOT 11.06  ; 上料盒区域1感应
LD 44.08  ; #1上顶升气缸伸出
ANDNOT 1.00  ; #1满料盒到位感应
ANDNOT 11.06  ; 上料盒区域1感应
ORLD
TIMX(550) 0913 &10  ; #1上顶升气缸缩回延时
; rung 57: ********NG输送带电机动作****** / NG通道电机动作 要加放料时不动的条件
LD W19.10  ; 启动状态
OUT TR0
AND 45.07  ; 检漏电机走
OUT 44.10  ; 检漏NG电机启动
LD TR0
LD 48.06  ; 龙门升降回检漏NG放料位
AND W34.02  ; 龙门升降在测试NG位置
AND 34.10  ; 龙门升降在原始位置
LDNOT 48.06  ; 龙门升降回检漏NG放料位
ANDNOT W34.02  ; 龙门升降在测试NG位置
ORLD
ANDLD
AND 3.00  ; 检漏NG放料位有料感应
TIMX(550) 0853 &1  ; 检漏电机延时走
@AND T0853  ; 检漏电机延时走
SET 45.07  ; 检漏电机走
LD TR0
AND 45.07  ; 检漏电机走
TIMX(550) 0854 &25
LD TR0
AND T0854
RSET 45.07  ; 检漏电机走

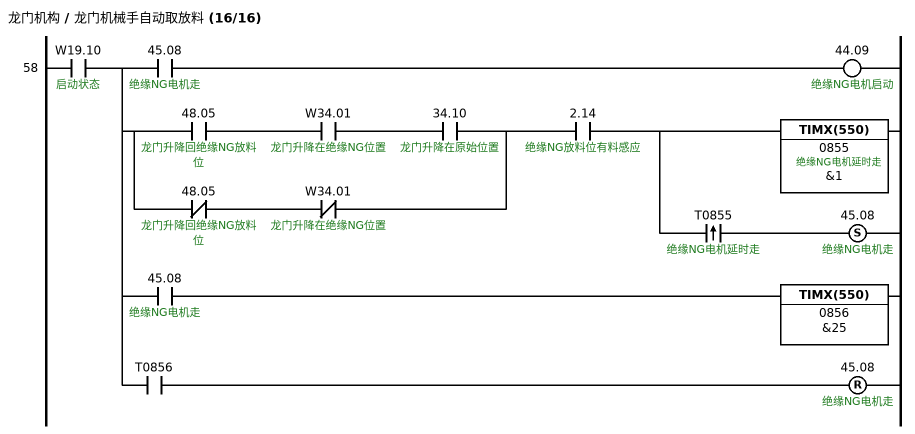
; rung 58
LD W19.10  ; 启动状态
OUT TR0
AND 45.08  ; 绝缘NG电机走
OUT 44.09  ; 绝缘NG电机启动
LD TR0
LD 48.05  ; 龙门升降回绝缘NG放料位
AND W34.01  ; 龙门升降在绝缘NG位置
AND 34.10  ; 龙门升降在原始位置
LDNOT 48.05  ; 龙门升降回绝缘NG放料位
ANDNOT W34.01  ; 龙门升降在绝缘NG位置
ORLD
ANDLD
AND 2.14  ; 绝缘NG放料位有料感应
TIMX(550) 0855 &1  ; 绝缘NG电机延时走
@AND T0855  ; 绝缘NG电机延时走
SET 45.08  ; 绝缘NG电机走
LD TR0
AND 45.08  ; 绝缘NG电机走
TIMX(550) 0856 &25
LD TR0
AND T0856
RSET 45.08  ; 绝缘NG电机走

### Section 龙门机构外部输出

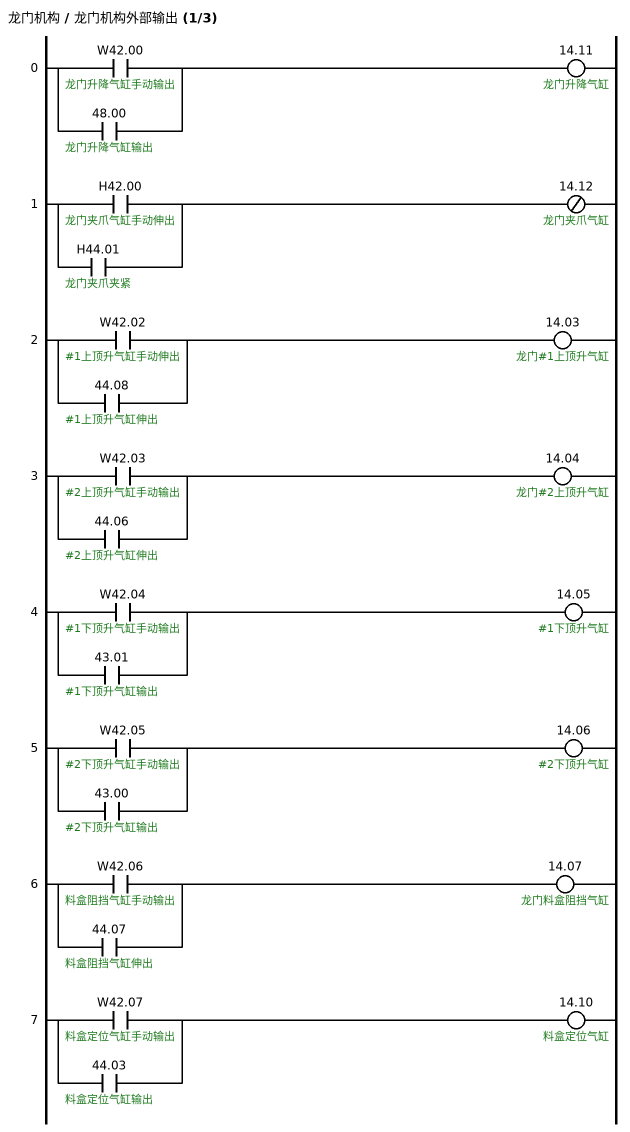
; rung 0
LD W42.00  ; 龙门升降气缸手动输出
OR 48.00  ; 龙门升降气缸输出
OUT 14.11  ; 龙门升降气缸
; rung 1
LD H42.00  ; 龙门夹爪气缸手动伸出
OR H44.01  ; 龙门夹爪夹紧
OUTNOT 14.12  ; 龙门夹爪气缸
; rung 2
LD W42.02  ; #1上顶升气缸手动伸出
OR 44.08  ; #1上顶升气缸伸出
OUT 14.03  ; 龙门#1上顶升气缸
; rung 3
LD W42.03  ; #2上顶升气缸手动输出
OR 44.06  ; #2上顶升气缸伸出
OUT 14.04  ; 龙门#2上顶升气缸
; rung 4
LD W42.04  ; #1下顶升气缸手动输出
OR 43.01  ; #1下顶升气缸输出
OUT 14.05  ; #1下顶升气缸
; rung 5
LD W42.05  ; #2下顶升气缸手动输出
OR 43.00  ; #2下顶升气缸输出
OUT 14.06  ; #2下顶升气缸
; rung 6
LD W42.06  ; 料盒阻挡气缸手动输出
OR 44.07  ; 料盒阻挡气缸伸出
OUT 14.07  ; 龙门料盒阻挡气缸
; rung 7
LD W42.07  ; 料盒定位气缸手动输出
OR 44.03  ; 料盒定位气缸输出
OUT 14.10  ; 料盒定位气缸

